Omron CX-Programmer project NewProject (CX-Programmer 9.73)

# PLC NewPLC1: CJ2M CPU12
I/O table (CPU CJ2M-CPU12): rack 0 slot 0 CJ1W-ID261; rack 0 slot 1 CJ1W-OD261; rack 0 slot 2 CJ1W-EIP21

## Global symbols (name address type ; comment)
AUTO 4030.00 BOOL  ; Auto
0.00 BOOL  ; (WP) SE Overload Product
0.01 BOOL  ; (HP) SE STOPPER SHIFTER
0.02 BOOL  ; (WP) SE STOPPER CHECKER 1
0.03 BOOL  ; (WP) SE STOPPER CHECKER 2
0.04 BOOL  ; (WP)SE NG PUSHER
0.05 BOOL  ; SE CHECKER 1
0.06 BOOL  ; SE CHECKER 2
0.07 BOOL  ; SE INPUT COUNT
0.08 BOOL  ; SE PRODUCT SHIFTER
0.09 BOOL  ; SE PRODUCT CHECKER 1
0.10 BOOL  ; SE PRODUCT CHECKER 2
0.11 BOOL  ; SE NG COUNT
0.12 BOOL  ; SE OUTPUT COUNT
0.13 BOOL  ; HP OVERLOAD PRODUCT
0.14 BOOL  ; WP OVERLOAD PRODUCT
0.15 BOOL  ; WP STOPPER SHIFTER
1.00 BOOL  ; WP STOPPER SHIFTER
1.01 BOOL  ; HP STOPPER CHECKER 1
1.02 BOOL  ; WP STOPPER CHECKER 1
1.03 BOOL  ; HP STOPPER CHECKER 2
1.04 BOOL  ; WP STOPPER CHECKER 2
1.05 BOOL  ; HP NG PUSHER
1.06 BOOL  ; WP NG PUSHER
1.07 BOOL  ; HP DOOR NG PRODUCT
1.08 BOOL  ; WP DOOR NG PRODUCT
1.09 BOOL  ; HP CHECKER 1
1.10 BOOL  ; WP CHECKER 1
1.11 BOOL  ; HP CHECKER 2
1.12 BOOL  ; WP CHECKER 2
1.13 BOOL  ; HP HORIZONTAL SHIFTER
1.14 BOOL  ; WP HORIZONTAL SHIFTER
1.15 BOOL  ; HP VERTICAL SHIFTER
2.00 BOOL  ; WP VERTICAL SHIFTER
2.01 BOOL  ; SE DOOR 1
2.02 BOOL  ; SE DOOR 2
2.03 BOOL  ; SE DOOR 3
2.04 BOOL  ; SE DOOR 4
2.05 BOOL  ; PB START 2
2.06 BOOL  ; PB START 1
2.07 BOOL  ; PB EXECUTE
2.08 BOOL  ; SE CHECKER 1 (2)
2.09 BOOL  ; SE CHECKER 1 (2)
2.15 BOOL  ; Pressure Sensor
300.00 BOOL  ; Hole Check Error
3070.00 BOOL  ; ALL HP TRANSFER
3070.01 BOOL  ; ALL HP CHECKER 1
3070.02 BOOL  ; ALL HP CHECKER 2
3070.03 BOOL  ; ALL HP NG EJECTOR
350.00 BOOL  ; U0_X_At_POS-0
350.01 BOOL  ; U0_X_At_POS-1
350.15 BOOL  ; U0_X_At_HOMEPOS
3.00 BOOL  ; AUTO BUTTON 1
3.01 BOOL  ; AUTO BUTTON 2
3.04 BOOL  ; DOOR SWITCH 1
3.05 BOOL  ; DOOR SWITCH 2
3.06 BOOL  ; DOOR SWITCH 3
3.07 BOOL  ; SE Minimum
3.08 BOOL  ; HP SEPARATOR 1
3.09 BOOL  ; HP SEPARATOR 2
3.10 BOOL  ; WP HOLDER
4000.00 BOOL  ; ON ON
4004.03 BOOL  ; FLG
4004.04 BOOL  ; BUSY
4004.05 BOOL  ; OR
4004.06 BOOL  ; RUN
4004.07 BOOL  ; ERROR
400.00 BOOL  ; TRANSFER_EMG_ALM
400.01 BOOL  ; CHECKER 1_EMG_ALM
400.02 BOOL  ; CHECKER 2 EMG_ALM
400.03 BOOL  ; NG EJECTOR_EMG_ALM
400.04 BOOL  ; 094 : Error Silinder NG Pusher
400.05 BOOL  ; 095 : Error Silinder Checker 1
400.06 BOOL  ; 096 : Error Silinder Checker 2
400.07 BOOL  ; 097 : Error Silinder Horizontral Shifter
400.08 BOOL  ; 098 : Error Silinder Vertical Shifter
400.09 BOOL  ; 099 : Error Silinder Door NG
400.15 BOOL  ; Transfer_EMG_Alarm
4010.00 BOOL  ; All Unit Ready
4010.01 BOOL  ; ALL CYL HP
4010.02 BOOL  ; NC Unit Error
4010.03 BOOL  ; ALL UNIT ORIGIN
4010.04 BOOL  ; ALL Manual OFF
4010.05 BOOL  ; ALL NO ALARM
4010.06 BOOL  ; Door Closed
4010.09 BOOL  ; Door Closed
4010.10 BOOL  ; READY Under RUN
4010.11 BOOL  ; READY AUTO START
4010.12 BOOL  ; ErrorReset Switch DU
401.00 BOOL  ; 090 : Error Silinder Holder Shifter (SE013/014) - Transfer
401.01 BOOL  ; 091 : Error Silinder Stopper Shifter (SE015/100) - Transfer
401.03 BOOL  ; 093 : Error Silinder Stopper Checker 2 (SE103/104) - Checking 2
401.04 BOOL  ; 094 : Error Silinder NG Pusher (SE105/106) - NG Ejector
401.05 BOOL  ; 095 : Error Silinder Checker 1 (SE109/110) - Checking 1
401.06 BOOL  ; 096 : Error Silinder Checker 2 (SE111/112) - Checking 2
401.07 BOOL  ; 097 : Error Silinder Horizontral Shifter (SE113/114) - Transfer
401.08 BOOL  ; 098 : Error Silinder Vertical Shifter (SE115/200) - Transfer
401.09 BOOL  ; 099 : Error Silinder Door NG (SE107/108) - NG Ejector
401.15 BOOL  ; Transfer ALM
4020.00 BOOL  ; Auto Index - Stop Lock
402.00 BOOL  ; 092 : Error Silinder Stopper Checker 1 (SE101/102) - Checking 1
402.00 BOOL  ; 092 : Error Silinder Stopper Checker 1
402.01 BOOL  ; 095 : Error Silinder Checker 1 (SE109/110) - Checking 1
402.15 BOOL  ; Checker 1 ALM
4030.00 BOOL  ; AUTO
4030.01 BOOL  ; STOP LOCK
4030.02 BOOL  ; STOP
4030.03 BOOL  ; Force STOP
4030.04 BOOL  ; Normal Run
4030.05 BOOL  ; Active Dry Run
4030.10 BOOL  ; Auto OFF
4031.00 BOOL  ; AUTO RUN PROCESS
4031.01 BOOL  ; SENSOR WORKING CHECK
4031.02 BOOL  ; SHIFT DATA UNIT WORK
4031.03 BOOL  ; START - AFTER CONFIRM
4031.04 BOOL  ; AUTO SAME START
4031.05 BOOL  ; AUTO DIFFERENT START
4031.06 BOOL  ; START Again
4031.07 BOOL  ; ReSTART Condition
4032.00 BOOL  ; AUTO - Transfer
4032.15 BOOL  ; FIN - Transfer
4033.00 BOOL  ; AUTO - Checker 1
4033.15 BOOL  ; FIN - Checker 1
4034.00 BOOL  ; AUTO - CHECKER 2
4034.15 BOOL  ; FIN - Checker 2
4035.00 BOOL  ; AUTO - NG EJECTOR
4035.04 BOOL  ; ACTIVE TYPE NON K
4035.05 BOOL  ; Active TYPE K
4035.15 BOOL  ; FIN - NG EJECTOR
4036.15 BOOL  ; FIN - Unloading
403.00 BOOL  ; 093 : Error Silinder Stopper Checker 2 (SE103/104) - Checking 2
403.01 BOOL  ; 096 : Error Silinder Checker 2 (SE111/112) - Checking 2
403.15 BOOL  ; Checker 2 ALM
4045.15 BOOL  ; ALL UNIT FINISH
4047.00 BOOL  ; Auto CL
4047.01 BOOL  ; Manu CL
4047.02 BOOL  ; RUN CLEAR LOAD
4047.03 BOOL  ; After Manual CL
404.00 BOOL  ; 094 : Error Silinder NG Pusher (SE105/106) - NG Ejector
404.01 BOOL  ; 099 : Error Silinder Door NG (SE107/108) - NG Ejector
404.09 BOOL  ; 099 : Error Silinder Door NG (SE107/108) - NG Ejector
404.15 BOOL  ; NG Ejector ALM
4050.00 BOOL  ; ALL EMPTY
4050.01 BOOL  ; ALL UNIT EMPTY
4050.02 BOOL  ; WORK - No Unit
4050.03 BOOL  ; WORK - Marking
4050.04 BOOL  ; WORK - No Unit
4050.05 BOOL  ; WORK - Unloading
4051.01 BOOL  ; All Unit Empty
4055.00 BOOL  ; Active Checker 1
4055.01 BOOL  ; Active No Unit
4055.02 BOOL  ; Active Checker 2
4055.03 BOOL  ; Active NG EJECTOR
4055.04 BOOL  ; Active NG STOPPER
4055.05 BOOL  ; Active Unloading
4056.00 BOOL  ; Active By Pass
405.00 BOOL  ; 095 : Error Silinder Checker 1
4060.10 BOOL  ; Fullwork
406.00 BOOL  ; 096 : Error Silinder Checker 2
4070.00 BOOL  ; EMG ALARM M/C
4070.01 BOOL  ; CYCLE ALARM M/C
4070.02 BOOL  ; NC UNIT ERROR
4076.03 BOOL  ; Active Marking No Part
407.00 BOOL  ; 097 : Error Silinder Horizontal Shifter
4080.00 BOOL  ; WAITING TIME
4081.00 BOOL  ; FULLWORK
4082.00 BOOL  ; BLOWING ON AFTER WAITING 2SEC
408.00 BOOL  ; 098 : Error Silinder Vertical Shifter
409.00 BOOL  ; 099 : Error Sillinder Door NG
4100.00 BOOL  ; Ready Transfer
4100.03 BOOL  ; Ready NG Stopper
4101.15 BOOL  ; DONE ORG Shifter Transfer
410.00 BOOL  ; Safety Door Alarm
4110.00 BOOL  ; POS 0 - Shifter Trasnfer
4110.01 BOOL  ; Pos 1 - Shifter Transfer
4110.15 BOOL  ; Home - Shifter Transfer
411.00 BOOL  ; 100 : Error Safety Door Front L (SE201) - Transfer
411.01 BOOL  ; 101 : Error Safety Door Front R (SE202) - Transfer
411.02 BOOL  ; 102 : Error Safety Door Back L (SE203) - Transfer
411.03 BOOL  ; 103 : Error Safety Door Back R (SE204) - Transfer
4120.00 BOOL  ; 1 Cycle Checking 1 (MANU)
4120.01 BOOL  ; Call Separator Seq
4120.05 BOOL  ; Ready Transfer
4121.00 BOOL  ; 1 Cycle Checking 2 (MANU)
4121.01 BOOL  ; Stopper On
4121.02 BOOL  ; Separator 1 On
4121.03 BOOL  ; Separator Off
4121.04 BOOL  ; Stopper Off
4121.11 BOOL  ; Stop Conv
4121.12 BOOL  ; On Conv
4121.15 BOOL  ; Finish Separator Seq
4122.00 BOOL  ; 1 Cycle Transfer (MANU)
4122.01 BOOL  ; Call Shifter
4123.00 BOOL  ; 1 Cycle NG Stopper (MANU)
4123.01 BOOL  ; Arm On
4123.02 BOOL  ; Separator 2 On
4123.03 BOOL  ; Shifter On
4123.04 BOOL  ; Arm Off
4123.05 BOOL  ; Separator 2 Off
4123.06 BOOL  ; Shifter Off
4123.10 BOOL  ; DONE - Transfer
4123.15 BOOL  ; Finish Shifter Seq
4124.00 BOOL  ; Status for Arm Down
4125.00 BOOL  ; 1 Cycle Checking NG
4126.00 BOOL  ; 1 Cycle NG Stopper (MANU)
4129.00 BOOL  ; 1 Cycle Process
412.00 BOOL  ; 104 : Error Low Air Pressure (SE215) - Transfer
4132.00 BOOL  ; MANUAL OFF
4140.00 BOOL  ; Anchor A_EMG_Error
4140.01 BOOL  ; Anchor A Error
4141.00 BOOL  ; 090 : Error Stopper (SE0100/0101) - Anchor A
4141.01 BOOL  ; 091 : Error Fwd/Bwd (SE0102/0103) - Anchor A
4141.02 BOOL  ; 092 : Error Rotary Esc (SE0104/0105) - Anchor A
4141.03 BOOL  ; 093 : Error Chuck PNP (SE0110) - Anchor A
4141.04 BOOL  ; 094 : Error Up/Dn Pusher (SE0111/0112) - Anchor A
4141.05 BOOL  ; 095 : Error Lift Case (SE0001/0002) - Anchor A
4141.06 BOOL  ; 096 : Error Holder Case (SE00114/00115) - Anchor A
4143.00 BOOL  ; 110 : Alarm Driver X Axis SMC - Anchor A
4143.01 BOOL  ; 111: Alarm Driver Y Axis SMC - Anchor A
4143.02 BOOL  ; 112 : Alarm Driver Rotary ARD K - Anchor A
4170.00 BOOL  ; Ready Transfer
4170.05 BOOL  ; Ready - Check HV
4172.10 BOOL  ; DONE - Check HV
4182.00 BOOL  ; Check HV Manu = OFF
4190.00 BOOL  ; Ready Transfer
4190.01 BOOL  ; Ready Checker 1
4190.02 BOOL  ; Ready Checker 2
4190.03 BOOL  ; Ready NG Stopper
4193.00 BOOL  ; Ready Transfer
4193.01 BOOL  ; Ready Checker 1
4193.02 BOOL  ; Ready Checker 2
4193.03 BOOL  ; Ready NG Stopper
4220.05 BOOL  ; Ready - Check CR
4221.15 BOOL  ; Finish Check CR
4222.10 BOOL  ; DONE - Check CR
4232.00 BOOL  ; Check CR Manu = OFF
4240.00 BOOL  ; Check CR_EMG_ALM
4240.01 BOOL  ; Check CR ALM
4270.05 BOOL  ; Ready - Marking
4282.00 BOOL  ; Marking Unit Manu = OFF
4290.00 BOOL  ; Marking Unit_EMG_ALM
4290.01 BOOL  ; Marking Unit ALM
4301.15 BOOL  ; DONE ORG Shifter Transfer
4320.05 BOOL  ; Ready - Unloading
4321.06 BOOL  ; Chuck Off
4324.00 BOOL  ; OK
4332.00 BOOL  ; Unloading Manu = OFF
4340.00 BOOL  ; Unloading_EMG_ALM
4340.01 BOOL  ; Unloading ALM
4390.00 BOOL  ; SafetyDoor_EMG_ALM
4390.01 BOOL  ; Safety Door ALM
4391.00 BOOL  ; Safety Door Front L
4391.01 BOOL  ; Safety Door Front C
4391.02 BOOL  ; Safety Door Front R
4391.03 BOOL  ; Safety Door Back L
4520.01 BOOL  ; Call START Check Hole 1
4520.02 BOOL  ; Call START Check Hole 2
4520.03 BOOL  ; Call NG
4520.15 BOOL  ; Finish Separator
4521.00 BOOL  ; START Check Hole 1
4521.01 BOOL  ; Holder 1 ON
4521.02 BOOL  ; Checker 1 DOWN
4521.03 BOOL  ; Checker 1 UP
4521.04 BOOL  ; Holder 1 OFF
4521.05 BOOL  ; CHECKER 2 ON
4521.06 BOOL  ; CHECKER 2 DOWN
4521.07 BOOL  ; CHECKER 2 UP
4521.08 BOOL  ; CHECKER 2 OFF
4521.10 BOOL  ; DONE - Checker 1
4521.15 BOOL  ; FINISH Check 1
4522.01 BOOL  ; Call Shifter
4523.00 BOOL  ; Start Shifter Seq
4523.01 BOOL  ; ARM VERTICAL ON
4523.02 BOOL  ; STOPPER ON
4523.03 BOOL  ; SHIFTER HORIZONTAL ON
4523.04 BOOL  ; ARM VERTICAL OFF
4523.05 BOOL  ; STOPPER OFF
4523.06 BOOL  ; SHIFTER HORIZONTAL OFF
4523.10 BOOL  ; DONE - Transfer
4523.15 BOOL  ; Finish Shifter Seq
4524.00 BOOL  ; START Check Hole 2
4524.01 BOOL  ; Holder 2 ON
4524.02 BOOL  ; Checker 2 DOWN
4524.03 BOOL  ; Checker 2 UP
4524.04 BOOL  ; Holder 2 OFF
4524.10 BOOL  ; DONE - Checker 2
4524.15 BOOL  ; FINISH Check 2
4525.00 BOOL  ; Start NG Seq
4525.01 BOOL  ; NG Door Down
4525.02 BOOL  ; NG Pusher ON
4525.03 BOOL  ; NG Pusher OFF
4525.04 BOOL  ; NG Door UP
4525.10 BOOL  ; DONE - NG EJECTOR
4525.15 BOOL  ; Finish NG Stopper Seq
4526.00 BOOL  ; Start NG Seq
4526.01 BOOL  ; NG Door DOWN
4526.02 BOOL  ; NG Pusher ON
4526.03 BOOL  ; NG Pusher OFF
4526.04 BOOL  ; NG Door UP
4526.15 BOOL  ; Finish NG Stopper Seq
4527.00 BOOL  ; Call Holder Seq
4527.01 BOOL  ; Holder On
4527.02 BOOL  ; Holder Off
4527.15 BOOL  ; Finish Seq Holder
4530.00 BOOL  ; START VISION 1 SEQ
4530.01 BOOL  ; MEASURE START VIS 1
4530.02 BOOL  ; MEASURE BUSY VIS 1
4530.03 BOOL  ; MEASURE FINISH VIS 1
4530.04 BOOL  ; JUDGE MEASURED
4530.15 BOOL  ; FINISH VISION 1
4531.00 BOOL  ; START VISION 2 SEQ
4531.01 BOOL  ; MEASURE START VIS 2
4531.02 BOOL  ; MEASURE BUSY VIS 2
4531.03 BOOL  ; MEASURE FINISH VIS 2
4531.04 BOOL  ; JUDGE MEASURED VIS 2
4531.05 BOOL  ; HOLDER OPEN VIS 2
4531.15 BOOL  ; FINISH VISION 2
4560.00 BOOL  ; Manual Transfer Active
4560.01 BOOL  ; Manual Checking 1 Active
4560.02 BOOL  ; Manual Checking 2 Active
4560.03 BOOL  ; Manual NG Ejector ACTIVE
4626.00 BOOL  ; Display OK/NG
4670.00 BOOL  ; PASSWORD CORRECT
4671.00 BOOL  ; Password SHOWUP
468.00 BOOL  ; TES
4725.00 BOOL  ; BLOWING ON
4725.01 BOOL  ; RUN 1x
4800.00 BOOL  ; Ready Transfer
4.00 BOOL  ; Silinder Overload Product
4.01 BOOL  ; Silinder Stopper Shifter
4.02 BOOL  ; Silinder Stopper Checker 1
4.03 BOOL  ; Silinder Stopper Checker 2
4.04 BOOL  ; Silinder NG Pusher
4.05 BOOL  ; Silinder Checker 1 DOWN
4.06 BOOL  ; Silinder Checker 1 UP
4.07 BOOL  ; Silinder Horizontal Shifter
4.08 BOOL  ; Silinder Vertical Shifter
4.09 BOOL  ; Silinder Door NG Product
4.10 BOOL  ; Buzzer
4.11 BOOL  ; Lamp PB Execute
4.12 BOOL  ; Lamp PB Start 1
4.13 BOOL  ; Air Pressure
4.14 BOOL  ; Lamp Red
4.15 BOOL  ; Lamp Green
5001.00 BOOL  ; Home Marking
500.00 BOOL  ; SILINDER OVERLOAD PRODUCT
500.01 BOOL  ; SILINDER STOPPER SHIFTER
500.02 BOOL  ; SILINDER STOPPER CHECKER 1
500.03 BOOL  ; SILINDER STOPPER CHECKER 2
500.04 BOOL  ; SILINDER NG PUSHER
500.05 BOOL  ; CHECKER 1 U/D
500.06 BOOL  ; CHECKER 2 U/D
500.07 BOOL  ; SILINDER HORIZONTAL SHIFTER
500.08 BOOL  ; SILINDER VERTICAL SHIFTER
500.09 BOOL  ; SILINDER DOOR NG PRODUCT
500.10 BOOL  ; BUZZER
500.11 BOOL  ; LAMP PB EXECUTE
500.12 BOOL  ; LAMP PB START 1
500.13 BOOL  ; AIR PRESSURE START
500.14 BOOL  ; LAMP RED
500.15 BOOL  ; LAMP GREEN
5010.00 BOOL  ; Reset
501.00 BOOL  ; MOTOR 1
501.01 BOOL  ; MOTOR 2
501.02 BOOL  ; Checker 2 DOWN
501.03 BOOL  ; Checker 2 UP
501.04 BOOL  ; Overload
501.05 BOOL  ; STOP
501.07 BOOL  ; Pressure 1
501.10 BOOL  ; MOTOR 2
501.15 BOOL  ; BLOWING
505.00 BOOL  ; Disable Marking
5.00 BOOL  ; Motor 1
5.01 BOOL  ; Motor 2
5.02 BOOL  ; Silinder Checker 2 DOWN
5.03 BOOL  ; Silinder Checker 2 UP
5.14 BOOL  ; NG DOOR LOCK
5.15 BOOL  ; BLOWING
645.00 BOOL  ; Reset Man CL
6.00 BOOL  ; WAITING TIME
700.00 BOOL  ; NG Check 1
70.00 BOOL  ; NG CHECK 1
760.00 BOOL  ; U/D  Checker 1
761.00 BOOL  ; U/D Checker 2
765.00 BOOL  ; Target Achieve
766.00 BOOL  ; NO TARGET
87.00 BOOL  ; Latch Main
D110 CHANNEL  ; Hasil Perhitungan EFF M/C
D11000 CHANNEL  ; Total Alarm Time
D120 CHANNEL  ; TOTAL OUTPUT OK+NG
D123 CHANNEL  ; CT M/C on Process
D124 CHANNEL  ; Output Target CT 1.5
D131 CHANNEL  ; Theoretical CT
D160 CHANNEL  ; YIELD RATIO
D18251 CHANNEL  ; M/C Cycle Time
D18270 CHANNEL  ; Output
D18271 CHANNEL  ; Input
D18284 CHANNEL  ; M/C Efficiency
D19299 CHANNEL  ; $?St$Bk?_#[6] / $?St$Bk?_#[6]
D19900 CHANNEL  ; Auto Run (second)
D19999 CHANNEL  ; $?St$Bk?_#[7] / $?St$Bk?_#[7]
D20000 CHANNEL  ; Total Alarm
D21100 CHANNEL  ; STOP TIME (second)
D21200 CHANNEL  ; ALARM TIME (second)
D21300 CHANNEL  ; OUTPUT OK
D21400 CHANNEL  ; WAITING TIME ( SEC )
D21500 CHANNEL  ; OUTPUT NG
D21600 CHANNEL  ; FULLWORK TIME (SEC)
D250 CHANNEL  ; TYPE
D4000 CHANNEL  ; OVERLOAD
D4002 CHANNEL  ; STOPPER
D4004 CHANNEL  ; STOPPER CHECKER 1
D4006 CHANNEL  ; STOPPER CHECKER 2
D4008 CHANNEL  ; NG PUSHER
D4010 CHANNEL  ; CHECKER 1 U/D
D4012 CHANNEL  ; Horizontal Shifter
D4014 CHANNEL  ; Vertical Shifter
D4016 CHANNEL  ; DOOR NG
D4018 CHANNEL  ; CHECKER 2 U/D
D4020 CHANNEL  ; Overload
E0.07 BOOL  ; SE Part 2
H10.00 BOOL  ; WORK - Checking 1
H10.01 BOOL  ; WORK - No Unit
H10.02 BOOL  ; WORK - Checker 2
H10.03 BOOL  ; WORK - NG Stopper
H10.04 BOOL  ; WORK - NG STOPPER
H14.00 BOOL  ; Enable Unit Checker 1
H14.01 BOOL  ; Enable Unit Checker 2
H14.02 BOOL  ; Enable Unit NG Stopper
H14.04 BOOL  ; Enable Unit Unloading
H18.00 BOOL  ; TYPE K
H18.01 BOOL  ; TYPE NON-K
H20.00 BOOL  ; Data Part In
H21.00 BOOL  ; OUTPUT NG
H25.00 BOOL  ; Active By Pass
H25.01 BOOL  ; NORMAL MODE
H25.02 BOOL  ; DRY RUN MODE
H70.00 BOOL  ; NG CHECK 1
H70.01 BOOL  ; NG CHECK 2
H72.00 BOOL  ; NG CHECK 1 (2)
T0060 BOOL  ; TIM ERROR
T0125 BOOL  ; RESET 1 SEC
T0200 BOOL  ; WAITING TIME
T0520 BOOL  ; Auto Button
T0521 BOOL  ; Auto Index Delay Finish
T0530 BOOL  ; UNIT WORKING AFTER CONFIRM (Dont ZERO)
T0531 BOOL  ; Delay for Start Again
T0533 BOOL  ; Time START CL
T0534 BOOL  ; DIFFERENT START
T0750 BOOL  ; Delay Checker 1
T0751 BOOL  ; Delay Checker 2
W0.00 BOOL  ; (WP)SE Overload Product
W0.01 BOOL  ; (HP)SE STOPPER SHIFTER
W0.02 BOOL  ; (WP)SE STOPPER CHECKER 1
W0.03 BOOL  ; (WP)SE STOPPER CHECKER 2
W0.04 BOOL  ; (WP)SE NG PUSHER
W0.05 BOOL  ; SE CHECKER 1
W0.06 BOOL  ; SE CHECKER 2
W0.07 BOOL  ; SE INPUT COUNT
W0.08 BOOL  ; SE PRODUCT SHIFTER
W0.09 BOOL  ; SE PRODUCT CHECKER 1
W0.10 BOOL  ; SE PRODUCT  CHECKER 2
W0.11 BOOL  ; SE NG COUNT
W0.12 BOOL  ; SE OUTPUT COUNT
W0.13 BOOL  ; HP SILINDER OVERLOAD PRODUCT
W0.14 BOOL  ; WP SILINDER OVERLOAD PRODUCT
W0.15 BOOL  ; WP SILINDER STOPPER SHIFTER
W110.00 BOOL  ; PB SILINDER OVERLOAD PRODUCT
W110.01 BOOL  ; PB SILINDER STOPPER SHIFTER
W110.02 BOOL  ; PB SILINDER STOPPER CHECKER 1
W110.03 BOOL  ; PB SILINDER STOPPER CHECKER 2
W110.04 BOOL  ; PB SILINDER NG PUSHER
W110.05 BOOL  ; PB SILINDER CHECKER 1
W110.06 BOOL  ; PB SILINDER CHECKER 2
W110.07 BOOL  ; PB SILINDER HORIZONTAL SHIFTER
W110.08 BOOL  ; PB SILINDER VERTICAL SHIFTER
W110.09 BOOL  ; PB SILINDER DOOR NG PRODUCT
W110.10 BOOL  ; PB BUZZER
W110.11 BOOL  ; PB LAMP PB EXECUTE
W110.12 BOOL  ; PB LAMP PB START 1
W110.13 BOOL  ; PB AIR PRESSURE
W110.14 BOOL  ; PB LAMP RED
W110.15 BOOL  ; PB LAMP GREEN
W111.00 BOOL  ; PB MOTOR 1
W111.01 BOOL  ; PB MOTOR 2
W111.02 BOOL  ; PB BLOWING
W111.10 BOOL  ; PB MOTOR 2
W120.00 BOOL  ; NS 1 Cycle Checking 1 (MANU)
W121.00 BOOL  ; NS 1 Cycle Checking 2 (MANU)
W122.00 BOOL  ; NS 1 Cycle Transfer  (MANU)
W123.00 BOOL  ; NS 1 Cycle NG Stopper (MANU)
W15.00 BOOL  ; NB By Pass M/C
W1.00 BOOL  ; WP SILINDER STOPPER SHIFTER
W1.01 BOOL  ; HP SILINDER STOPPER CHECKER 1
W1.02 BOOL  ; WP SILINDER STOPPER CHECKER 1
W1.03 BOOL  ; HP SILINDER STOPPER CHECKER 2
W1.04 BOOL  ; WP SILINDER STOPPER CHECKER 2
W1.05 BOOL  ; HP SILINDER NG PUSHER
W1.06 BOOL  ; WP SILINDER NG PUSHER
W1.07 BOOL  ; HP SILINDER DOOR NG PRODUCT
W1.08 BOOL  ; WP SILINDER DOOR NG PRODUCT
W1.09 BOOL  ; HP SILINDER CHECKER 1
W1.10 BOOL  ; WP SILINDER CHECKER 1
W1.11 BOOL  ; HP SILINDER CHECKER 2
W1.12 BOOL  ; WP SILINDER CHECKER 2
W1.13 BOOL  ; HP SILINDER HORIZONTAL SHIFTER
W1.14 BOOL  ; WP SILINDER HORIZONTAL SHIFTER
W1.15 BOOL  ; HP SILINDER VERTICAL SHIFTER
W20.00 BOOL  ; MAIN SW
W2.00 BOOL  ; WP SILINDER VERTICAL SHIFTER
W2.01 BOOL  ; SE SAFETY DOOR 1 (Front L)
W2.02 BOOL  ; SE SAFETY DOOR 2 (Front R)
W2.03 BOOL  ; SE SAFETYDOOR 3 (Back L)
W2.04 BOOL  ; SE SAFETYDOOR 4 (Back R)
W2.05 BOOL  ; PB START 2
W2.06 BOOL  ; PB START 1
W2.07 BOOL  ; PB EXECUTE
W2.08 BOOL  ; SE CHECKER 1 (2)
W2.09 BOOL  ; SE CHECKER 1 (2)
W2.15 BOOL  ; PRESSURE SENSOR
W30.00 BOOL  ; NS AUTO RUN
W30.03 BOOL  ; NS Normal Run
W30.04 BOOL  ; NS Dry Run
W30.05 BOOL  ; Manu Clear Load
W35.03 BOOL  ; NS TYPE NON K
W35.04 BOOL  ; NS TYPE K
W3.00 BOOL  ; VIS 1 FLG
W3.01 BOOL  ; VIS1 BUSY
W3.02 BOOL  ; VIS1 OR
W3.03 BOOL  ; VIS 1 RUN
W3.04 BOOL  ; VIS 1 ERROR
W3.05 BOOL  ; VIS2 FLG
W3.06 BOOL  ; VIS2 BUSY
W3.07 BOOL  ; VIS2 OR
W3.08 BOOL  ; VIS2 RUN
W3.09 BOOL  ; VIS2 ERROR
W50.00 BOOL  ; NS Checking 1 Active
W50.01 BOOL  ; NS Checking 2 Active
W50.02 BOOL  ; NS NG Active
W50.03 BOOL  ; NS Checking Active
W50.04 BOOL  ; NS Take Out Active
W52.01 BOOL  ; Reset Start Interlock
W60.00 BOOL  ; STOP
W6.00 BOOL  ; WAITING TIME
W70.00 BOOL  ; NS Reset ALM
W70.01 BOOL  ; Reset Record
W70.02 BOOL  ; Reset Time Record
W71.00 BOOL  ; DISPLAY OK/NG
ERROR_RST 4010.12 BOOL  ; ErrorReset Switch DU
EXECUTE W10.00 BOOL
OFF CF114 BOOL  ; ALWAYS OFF
ON CF113 BOOL  ; ALWAYS ON
ON_ON 4000.00 BOOL
RESET W70.00 BOOL  ; NS Reset ALM
RST_RECORD W70.01 BOOL  ; Reset Record

## Program Main_Control (cyclic task 0)
Local symbols
First_On BOOL
ON CF113 BOOL
P_OFF BOOL
on BOOL

### Section Input

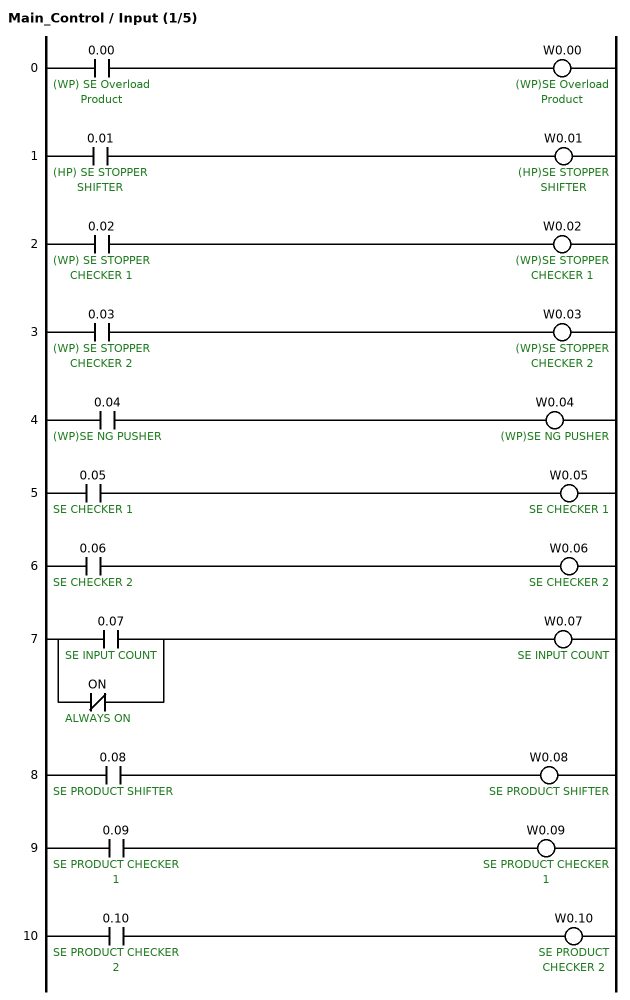
; rung 0
LD 0.00  ; (WP) SE Overload Product
OUT W0.00  ; (WP)SE Overload Product
; rung 1
LD 0.01  ; (HP) SE STOPPER SHIFTER
OUT W0.01  ; (HP)SE STOPPER SHIFTER
; rung 2
LD 0.02  ; (WP) SE STOPPER CHECKER 1
OUT W0.02  ; (WP)SE STOPPER CHECKER 1
; rung 3
LD 0.03  ; (WP) SE STOPPER CHECKER 2
OUT W0.03  ; (WP)SE STOPPER CHECKER 2
; rung 4
LD 0.04  ; (WP)SE NG PUSHER
OUT W0.04  ; (WP)SE NG PUSHER
; rung 5
LD 0.05  ; SE CHECKER 1
OUT W0.05  ; SE CHECKER 1
; rung 6
LD 0.06  ; SE CHECKER 2
OUT W0.06  ; SE CHECKER 2
; rung 7
LD 0.07  ; SE INPUT COUNT
ORNOT ON  ; ALWAYS ON
OUT W0.07  ; SE INPUT COUNT
; rung 8
LD 0.08  ; SE PRODUCT SHIFTER
OUT W0.08  ; SE PRODUCT SHIFTER
; rung 9
LD 0.09  ; SE PRODUCT CHECKER 1
OUT W0.09  ; SE PRODUCT CHECKER 1
; rung 10
LD 0.10  ; SE PRODUCT CHECKER 2
OUT W0.10  ; SE PRODUCT  CHECKER 2

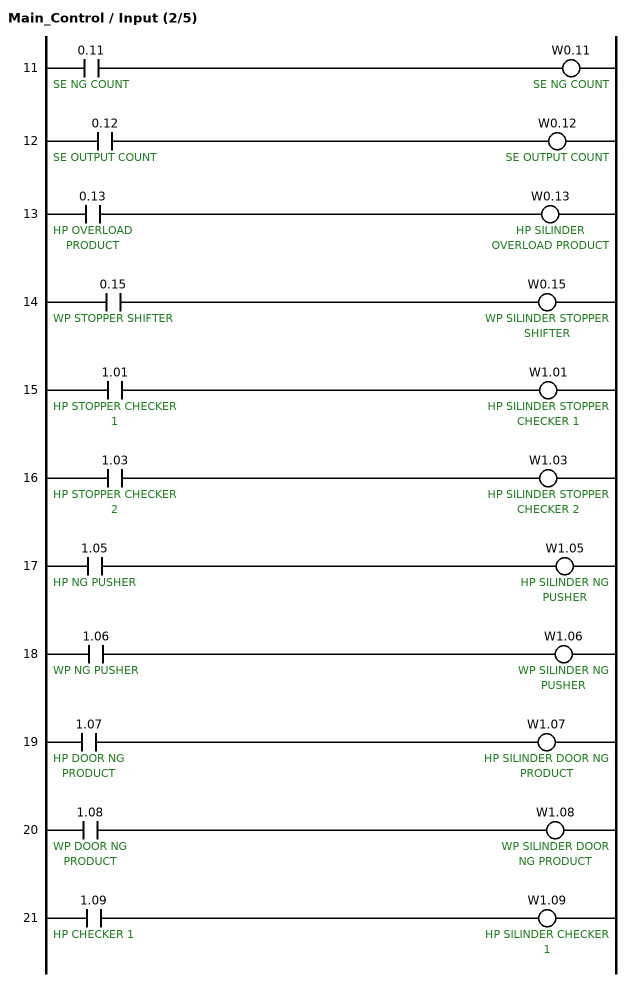
; rung 11
LD 0.11  ; SE NG COUNT
OUT W0.11  ; SE NG COUNT
; rung 12
LD 0.12  ; SE OUTPUT COUNT
OUT W0.12  ; SE OUTPUT COUNT
; rung 13
LD 0.13  ; HP OVERLOAD PRODUCT
OUT W0.13  ; HP SILINDER OVERLOAD PRODUCT
; rung 14
LD 0.15  ; WP STOPPER SHIFTER
OUT W0.15  ; WP SILINDER STOPPER SHIFTER
; rung 15
LD 1.01  ; HP STOPPER CHECKER 1
OUT W1.01  ; HP SILINDER STOPPER CHECKER 1
; rung 16
LD 1.03  ; HP STOPPER CHECKER 2
OUT W1.03  ; HP SILINDER STOPPER CHECKER 2
; rung 17
LD 1.05  ; HP NG PUSHER
OUT W1.05  ; HP SILINDER NG PUSHER
; rung 18
LD 1.06  ; WP NG PUSHER
OUT W1.06  ; WP SILINDER NG PUSHER
; rung 19
LD 1.07  ; HP DOOR NG PRODUCT
OUT W1.07  ; HP SILINDER DOOR NG PRODUCT
; rung 20
LD 1.08  ; WP DOOR NG PRODUCT
OUT W1.08  ; WP SILINDER DOOR NG PRODUCT
; rung 21
LD 1.09  ; HP CHECKER 1
OUT W1.09  ; HP SILINDER CHECKER 1

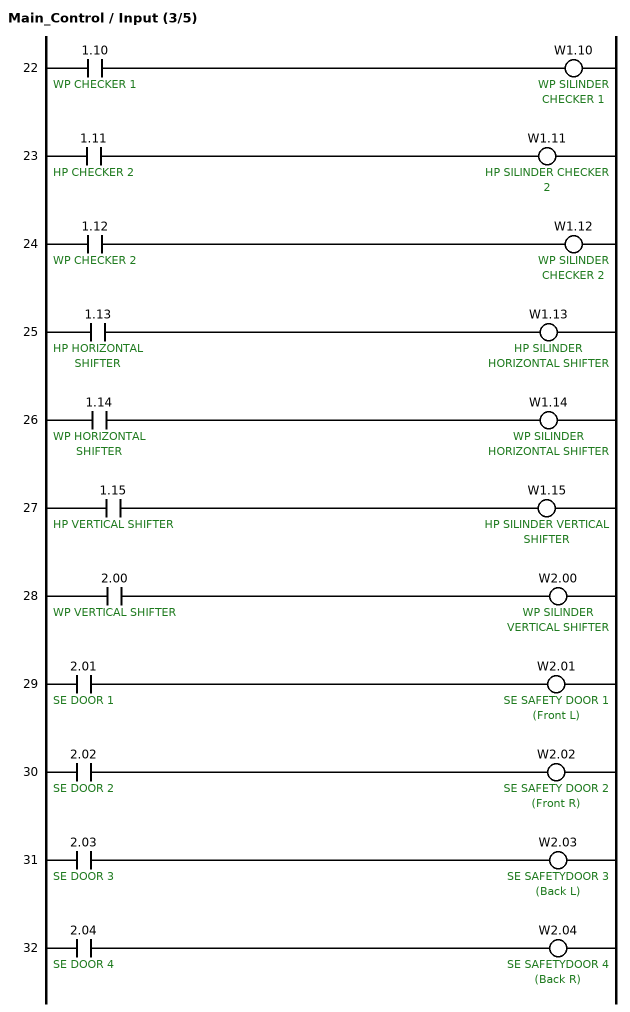
; rung 22
LD 1.10  ; WP CHECKER 1
OUT W1.10  ; WP SILINDER CHECKER 1
; rung 23
LD 1.11  ; HP CHECKER 2
OUT W1.11  ; HP SILINDER CHECKER 2
; rung 24
LD 1.12  ; WP CHECKER 2
OUT W1.12  ; WP SILINDER CHECKER 2
; rung 25
LD 1.13  ; HP HORIZONTAL SHIFTER
OUT W1.13  ; HP SILINDER HORIZONTAL SHIFTER
; rung 26
LD 1.14  ; WP HORIZONTAL SHIFTER
OUT W1.14  ; WP SILINDER HORIZONTAL SHIFTER
; rung 27
LD 1.15  ; HP VERTICAL SHIFTER
OUT W1.15  ; HP SILINDER VERTICAL SHIFTER
; rung 28
LD 2.00  ; WP VERTICAL SHIFTER
OUT W2.00  ; WP SILINDER VERTICAL SHIFTER
; rung 29
LD 2.01  ; SE DOOR 1
OUT W2.01  ; SE SAFETY DOOR 1 (Front L)
; rung 30
LD 2.02  ; SE DOOR 2
OUT W2.02  ; SE SAFETY DOOR 2 (Front R)
; rung 31
LD 2.03  ; SE DOOR 3
OUT W2.03  ; SE SAFETYDOOR 3 (Back L)
; rung 32
LD 2.04  ; SE DOOR 4
OUT W2.04  ; SE SAFETYDOOR 4 (Back R)

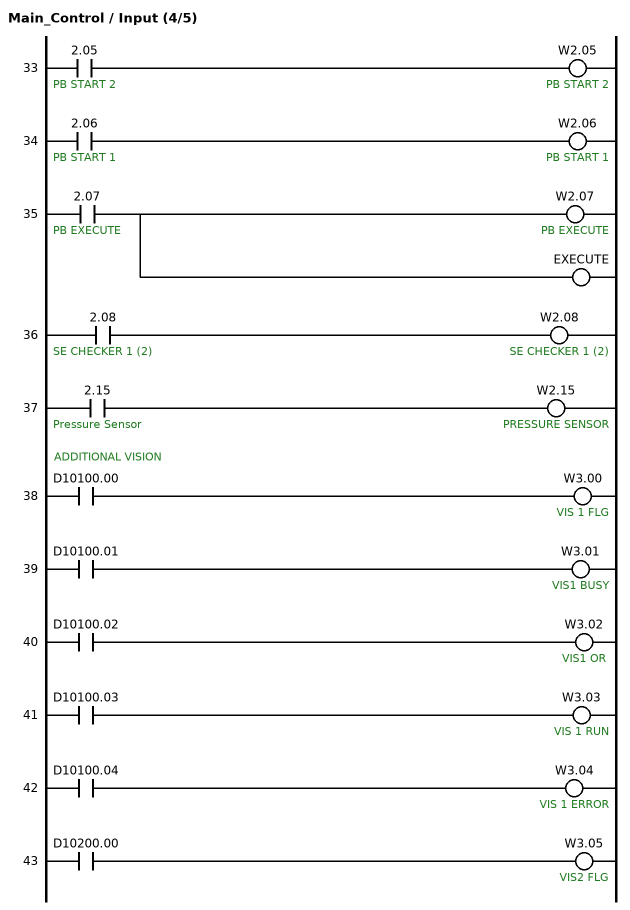
; rung 33
LD 2.05  ; PB START 2
OUT W2.05  ; PB START 2
; rung 34
LD 2.06  ; PB START 1
OUT W2.06  ; PB START 1
; rung 35
LD 2.07  ; PB EXECUTE
OUT W2.07  ; PB EXECUTE
OUT EXECUTE
; rung 36
LD 2.08  ; SE CHECKER 1 (2)
OUT W2.08  ; SE CHECKER 1 (2)
; rung 37
LD 2.15  ; Pressure Sensor
OUT W2.15  ; PRESSURE SENSOR
; rung 38: ADDITIONAL VISION
LD D10100.00
OUT W3.00  ; VIS 1 FLG
; rung 39
LD D10100.01
OUT W3.01  ; VIS1 BUSY
; rung 40
LD D10100.02
OUT W3.02  ; VIS1 OR
; rung 41
LD D10100.03
OUT W3.03  ; VIS 1 RUN
; rung 42
LD D10100.04
OUT W3.04  ; VIS 1 ERROR
; rung 43
LD D10200.00
OUT W3.05  ; VIS2 FLG

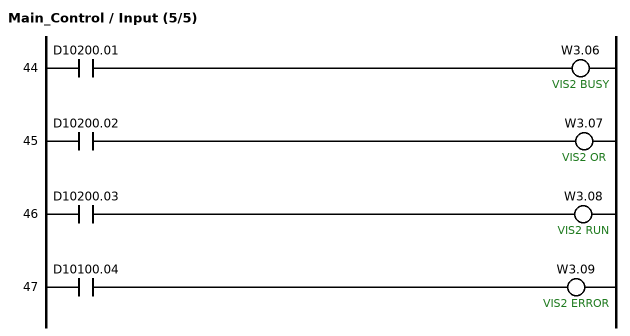
; rung 44
LD D10200.01
OUT W3.06  ; VIS2 BUSY
; rung 45
LD D10200.02
OUT W3.07  ; VIS2 OR
; rung 46
LD D10200.03
OUT W3.08  ; VIS2 RUN
; rung 47
LD D10100.04
OUT W3.09  ; VIS2 ERROR

### Section Output

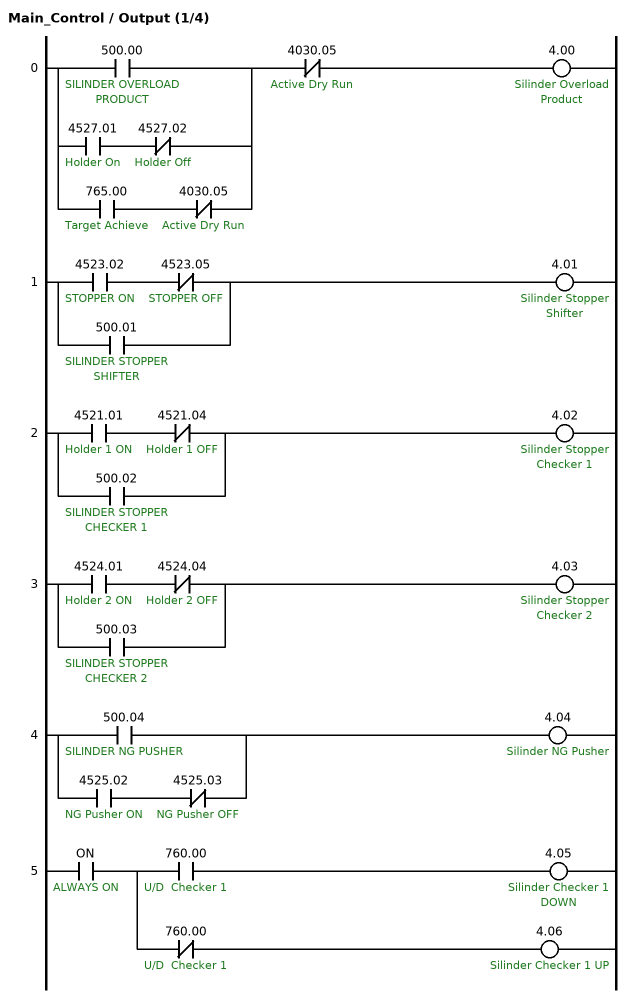
; rung 0
LD 500.00  ; SILINDER OVERLOAD PRODUCT
LD 4527.01  ; Holder On
ANDNOT 4527.02  ; Holder Off
ORLD
LD 765.00  ; Target Achieve
ANDNOT 4030.05  ; Active Dry Run
ORLD
ANDNOT 4030.05  ; Active Dry Run
OUT 4.00  ; Silinder Overload Product
; rung 1
LD 4523.02  ; STOPPER ON
ANDNOT 4523.05  ; STOPPER OFF
OR 500.01  ; SILINDER STOPPER SHIFTER
OUT 4.01  ; Silinder Stopper Shifter
; rung 2
LD 4521.01  ; Holder 1 ON
ANDNOT 4521.04  ; Holder 1 OFF
OR 500.02  ; SILINDER STOPPER CHECKER 1
OUT 4.02  ; Silinder Stopper Checker 1
; rung 3
LD 4524.01  ; Holder 2 ON
ANDNOT 4524.04  ; Holder 2 OFF
OR 500.03  ; SILINDER STOPPER CHECKER 2
OUT 4.03  ; Silinder Stopper Checker 2
; rung 4
LD 500.04  ; SILINDER NG PUSHER
LD 4525.02  ; NG Pusher ON
ANDNOT 4525.03  ; NG Pusher OFF
ORLD
OUT 4.04  ; Silinder NG Pusher
; rung 5
LD ON  ; ALWAYS ON
OUT TR0
AND 760.00  ; U/D  Checker 1
OUT 4.05  ; Silinder Checker 1 DOWN
LD TR0
ANDNOT 760.00  ; U/D  Checker 1
OUT 4.06  ; Silinder Checker 1 UP

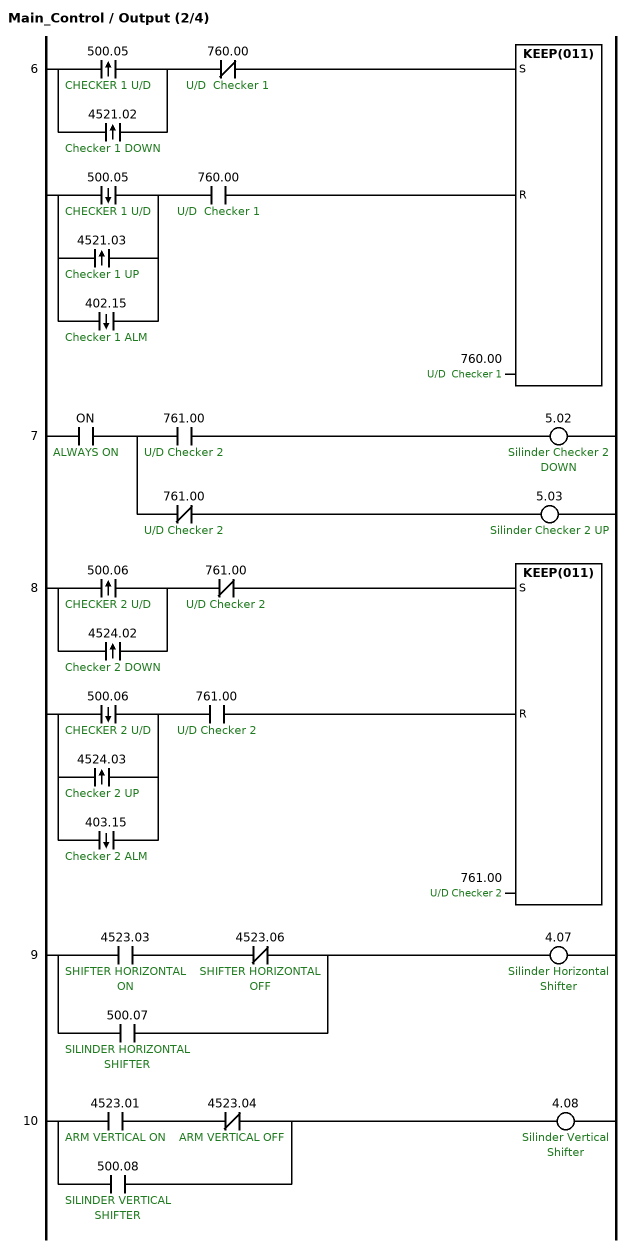
; rung 6
@LD 500.05  ; CHECKER 1 U/D
@OR 4521.02  ; Checker 1 DOWN
ANDNOT 760.00  ; U/D  Checker 1
%LD 500.05  ; CHECKER 1 U/D
@OR 4521.03  ; Checker 1 UP
%OR 402.15  ; Checker 1 ALM
AND 760.00  ; U/D  Checker 1
KEEP(011) 760.00  ; U/D  Checker 1
; rung 7
LD ON  ; ALWAYS ON
OUT TR0
AND 761.00  ; U/D Checker 2
OUT 5.02  ; Silinder Checker 2 DOWN
LD TR0
ANDNOT 761.00  ; U/D Checker 2
OUT 5.03  ; Silinder Checker 2 UP
; rung 8
@LD 500.06  ; CHECKER 2 U/D
@OR 4524.02  ; Checker 2 DOWN
ANDNOT 761.00  ; U/D Checker 2
%LD 500.06  ; CHECKER 2 U/D
@OR 4524.03  ; Checker 2 UP
%OR 403.15  ; Checker 2 ALM
AND 761.00  ; U/D Checker 2
KEEP(011) 761.00  ; U/D Checker 2
; rung 9
LD 4523.03  ; SHIFTER HORIZONTAL ON
ANDNOT 4523.06  ; SHIFTER HORIZONTAL OFF
OR 500.07  ; SILINDER HORIZONTAL SHIFTER
OUT 4.07  ; Silinder Horizontal Shifter
; rung 10
LD 4523.01  ; ARM VERTICAL ON
ANDNOT 4523.04  ; ARM VERTICAL OFF
OR 500.08  ; SILINDER VERTICAL SHIFTER
OUT 4.08  ; Silinder Vertical Shifter

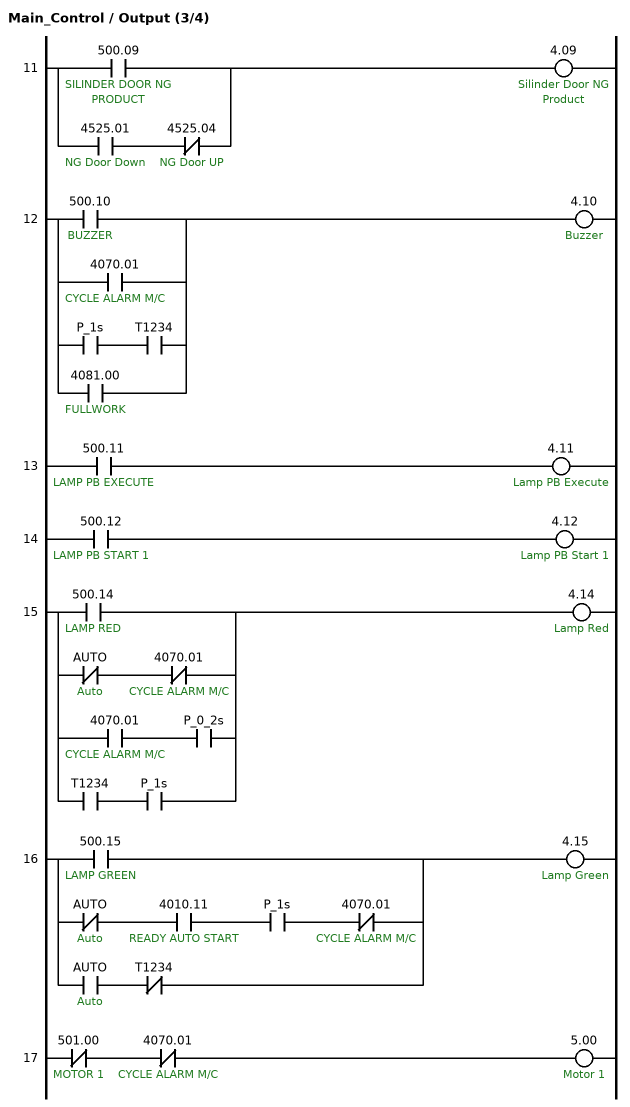
; rung 11
LD 500.09  ; SILINDER DOOR NG PRODUCT
LD 4525.01  ; NG Door Down
ANDNOT 4525.04  ; NG Door UP
ORLD
OUT 4.09  ; Silinder Door NG Product
; rung 12
LD 500.10  ; BUZZER
OR 4070.01  ; CYCLE ALARM M/C
LD P_1s
AND T1234
ORLD
OR 4081.00  ; FULLWORK
OUT 4.10  ; Buzzer
; rung 13
LD 500.11  ; LAMP PB EXECUTE
OUT 4.11  ; Lamp PB Execute
; rung 14
LD 500.12  ; LAMP PB START 1
OUT 4.12  ; Lamp PB Start 1
; rung 15
LD 500.14  ; LAMP RED
LDNOT AUTO  ; Auto
ANDNOT 4070.01  ; CYCLE ALARM M/C
ORLD
LD 4070.01  ; CYCLE ALARM M/C
AND P_0_2s
ORLD
LD T1234
AND P_1s
ORLD
OUT 4.14  ; Lamp Red
; rung 16
LD 500.15  ; LAMP GREEN
LDNOT AUTO  ; Auto
AND 4010.11  ; READY AUTO START
AND P_1s
ANDNOT 4070.01  ; CYCLE ALARM M/C
ORLD
LD AUTO  ; Auto
ANDNOT T1234
ORLD
OUT 4.15  ; Lamp Green
; rung 17
LDNOT 501.00  ; MOTOR 1
ANDNOT 4070.01  ; CYCLE ALARM M/C
OUT 5.00  ; Motor 1

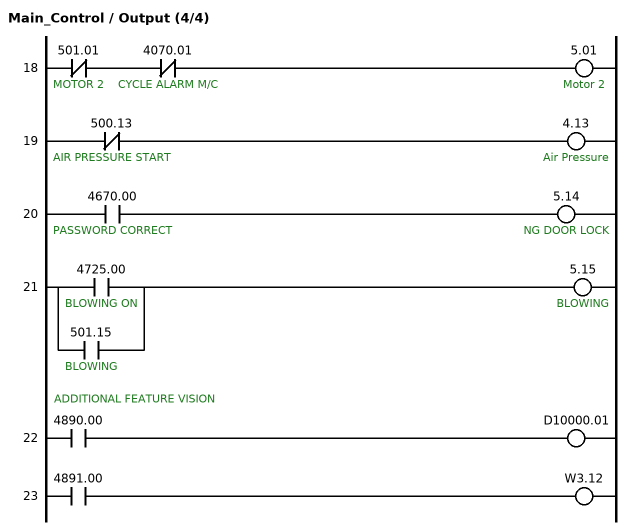
; rung 18
LDNOT 501.01  ; MOTOR 2
ANDNOT 4070.01  ; CYCLE ALARM M/C
OUT 5.01  ; Motor 2
; rung 19
LDNOT 500.13  ; AIR PRESSURE START
OUT 4.13  ; Air Pressure
; rung 20
LD 4670.00  ; PASSWORD CORRECT
OUT 5.14  ; NG DOOR LOCK
; rung 21
LD 4725.00  ; BLOWING ON
OR 501.15  ; BLOWING
OUT 5.15  ; BLOWING
; rung 22: ADDITIONAL FEATURE VISION
LD 4890.00
OUT D10000.01
; rung 23
LD 4891.00
OUT W3.12

### Section Manual

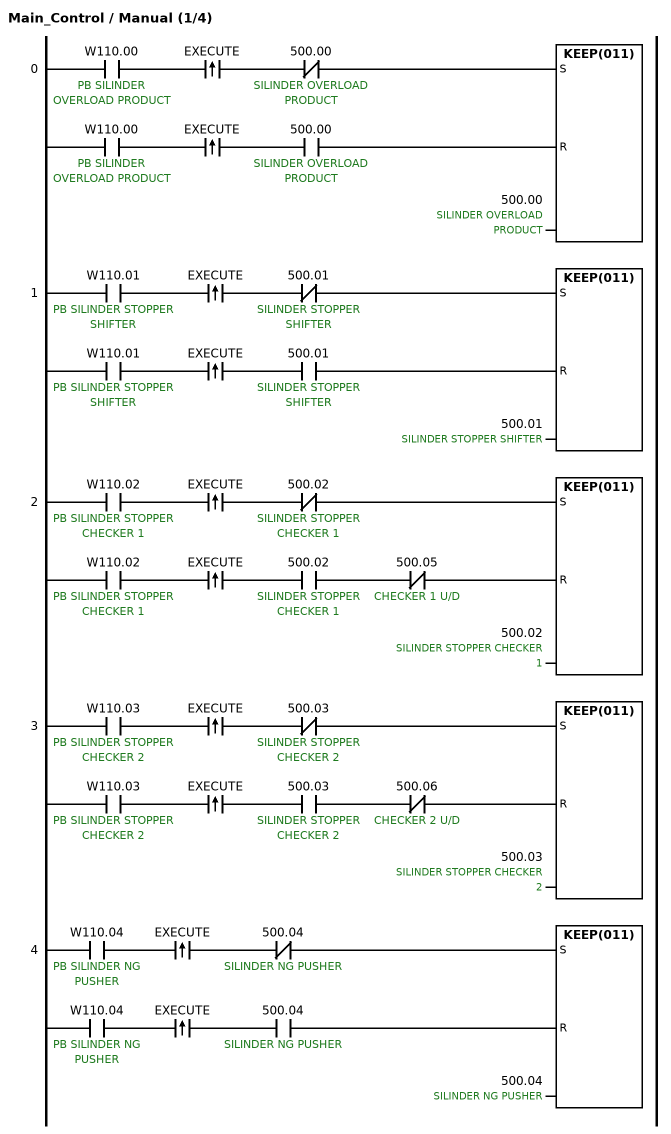
; rung 0
LD W110.00  ; PB SILINDER OVERLOAD PRODUCT
@AND EXECUTE
ANDNOT 500.00  ; SILINDER OVERLOAD PRODUCT
LD W110.00  ; PB SILINDER OVERLOAD PRODUCT
@AND EXECUTE
AND 500.00  ; SILINDER OVERLOAD PRODUCT
KEEP(011) 500.00  ; SILINDER OVERLOAD PRODUCT
; rung 1
LD W110.01  ; PB SILINDER STOPPER SHIFTER
@AND EXECUTE
ANDNOT 500.01  ; SILINDER STOPPER SHIFTER
LD W110.01  ; PB SILINDER STOPPER SHIFTER
@AND EXECUTE
AND 500.01  ; SILINDER STOPPER SHIFTER
KEEP(011) 500.01  ; SILINDER STOPPER SHIFTER
; rung 2
LD W110.02  ; PB SILINDER STOPPER CHECKER 1
@AND EXECUTE
ANDNOT 500.02  ; SILINDER STOPPER CHECKER 1
LD W110.02  ; PB SILINDER STOPPER CHECKER 1
@AND EXECUTE
AND 500.02  ; SILINDER STOPPER CHECKER 1
ANDNOT 500.05  ; CHECKER 1 U/D
KEEP(011) 500.02  ; SILINDER STOPPER CHECKER 1
; rung 3
LD W110.03  ; PB SILINDER STOPPER CHECKER 2
@AND EXECUTE
ANDNOT 500.03  ; SILINDER STOPPER CHECKER 2
LD W110.03  ; PB SILINDER STOPPER CHECKER 2
@AND EXECUTE
AND 500.03  ; SILINDER STOPPER CHECKER 2
ANDNOT 500.06  ; CHECKER 2 U/D
KEEP(011) 500.03  ; SILINDER STOPPER CHECKER 2
; rung 4
LD W110.04  ; PB SILINDER NG PUSHER
@AND EXECUTE
ANDNOT 500.04  ; SILINDER NG PUSHER
LD W110.04  ; PB SILINDER NG PUSHER
@AND EXECUTE
AND 500.04  ; SILINDER NG PUSHER
KEEP(011) 500.04  ; SILINDER NG PUSHER

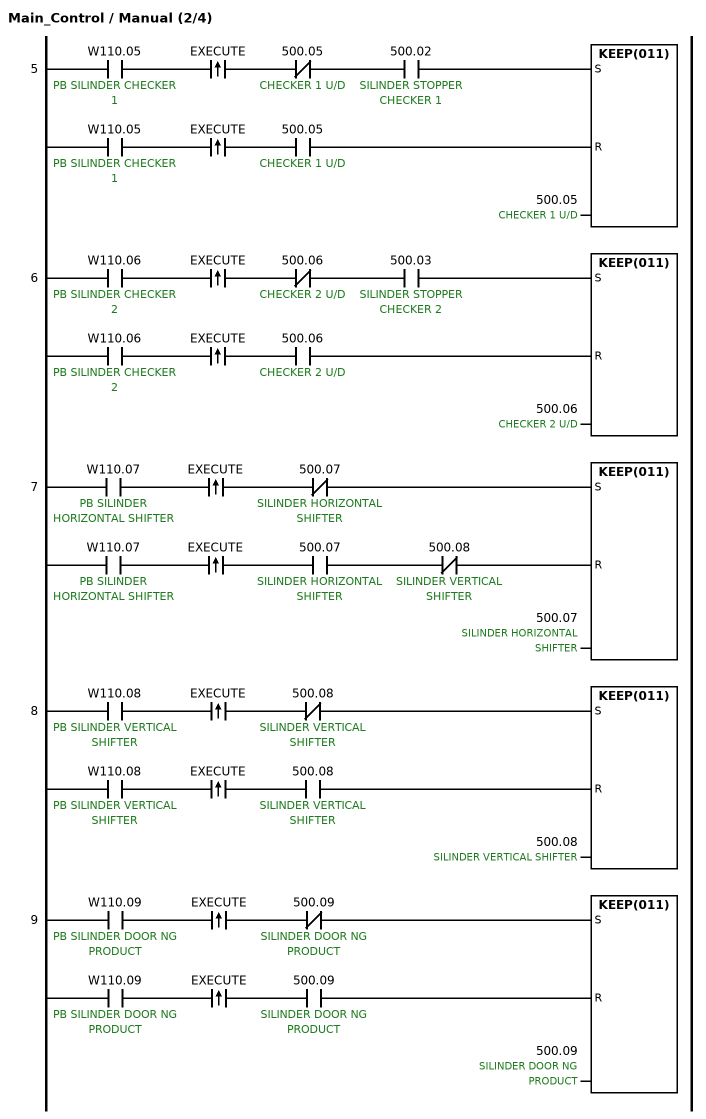
; rung 5
LD W110.05  ; PB SILINDER CHECKER 1
@AND EXECUTE
ANDNOT 500.05  ; CHECKER 1 U/D
AND 500.02  ; SILINDER STOPPER CHECKER 1
LD W110.05  ; PB SILINDER CHECKER 1
@AND EXECUTE
AND 500.05  ; CHECKER 1 U/D
KEEP(011) 500.05  ; CHECKER 1 U/D
; rung 6
LD W110.06  ; PB SILINDER CHECKER 2
@AND EXECUTE
ANDNOT 500.06  ; CHECKER 2 U/D
AND 500.03  ; SILINDER STOPPER CHECKER 2
LD W110.06  ; PB SILINDER CHECKER 2
@AND EXECUTE
AND 500.06  ; CHECKER 2 U/D
KEEP(011) 500.06  ; CHECKER 2 U/D
; rung 7
LD W110.07  ; PB SILINDER HORIZONTAL SHIFTER
@AND EXECUTE
ANDNOT 500.07  ; SILINDER HORIZONTAL SHIFTER
LD W110.07  ; PB SILINDER HORIZONTAL SHIFTER
@AND EXECUTE
AND 500.07  ; SILINDER HORIZONTAL SHIFTER
ANDNOT 500.08  ; SILINDER VERTICAL SHIFTER
KEEP(011) 500.07  ; SILINDER HORIZONTAL SHIFTER
; rung 8
LD W110.08  ; PB SILINDER VERTICAL SHIFTER
@AND EXECUTE
ANDNOT 500.08  ; SILINDER VERTICAL SHIFTER
LD W110.08  ; PB SILINDER VERTICAL SHIFTER
@AND EXECUTE
AND 500.08  ; SILINDER VERTICAL SHIFTER
KEEP(011) 500.08  ; SILINDER VERTICAL SHIFTER
; rung 9
LD W110.09  ; PB SILINDER DOOR NG PRODUCT
@AND EXECUTE
ANDNOT 500.09  ; SILINDER DOOR NG PRODUCT
LD W110.09  ; PB SILINDER DOOR NG PRODUCT
@AND EXECUTE
AND 500.09  ; SILINDER DOOR NG PRODUCT
KEEP(011) 500.09  ; SILINDER DOOR NG PRODUCT

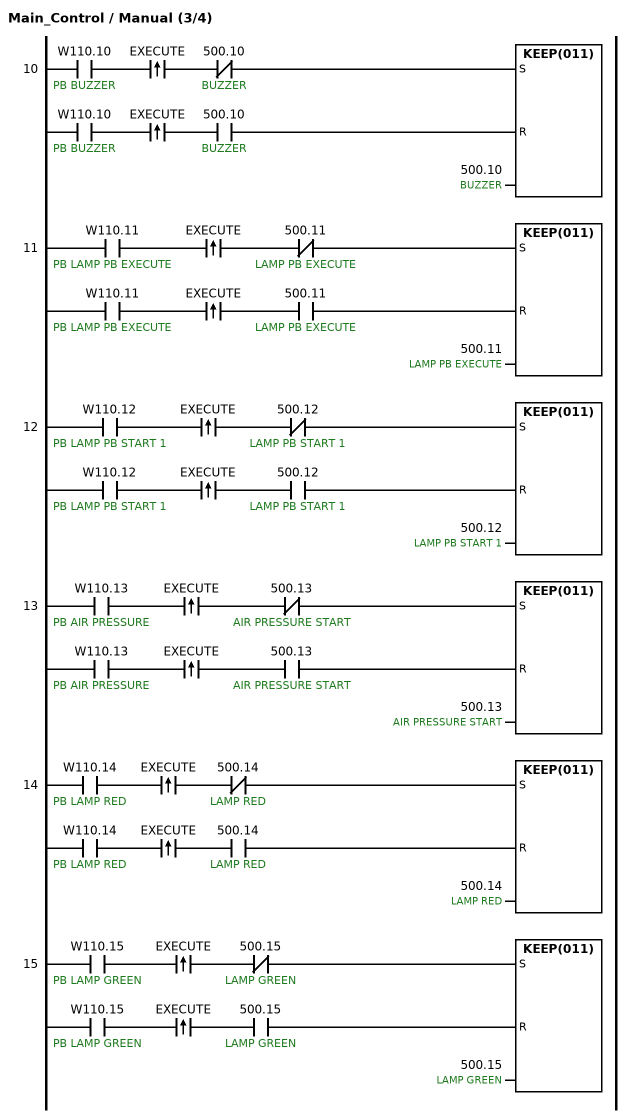
; rung 10
LD W110.10  ; PB BUZZER
@AND EXECUTE
ANDNOT 500.10  ; BUZZER
LD W110.10  ; PB BUZZER
@AND EXECUTE
AND 500.10  ; BUZZER
KEEP(011) 500.10  ; BUZZER
; rung 11
LD W110.11  ; PB LAMP PB EXECUTE
@AND EXECUTE
ANDNOT 500.11  ; LAMP PB EXECUTE
LD W110.11  ; PB LAMP PB EXECUTE
@AND EXECUTE
AND 500.11  ; LAMP PB EXECUTE
KEEP(011) 500.11  ; LAMP PB EXECUTE
; rung 12
LD W110.12  ; PB LAMP PB START 1
@AND EXECUTE
ANDNOT 500.12  ; LAMP PB START 1
LD W110.12  ; PB LAMP PB START 1
@AND EXECUTE
AND 500.12  ; LAMP PB START 1
KEEP(011) 500.12  ; LAMP PB START 1
; rung 13
LD W110.13  ; PB AIR PRESSURE
@AND EXECUTE
ANDNOT 500.13  ; AIR PRESSURE START
LD W110.13  ; PB AIR PRESSURE
@AND EXECUTE
AND 500.13  ; AIR PRESSURE START
KEEP(011) 500.13  ; AIR PRESSURE START
; rung 14
LD W110.14  ; PB LAMP RED
@AND EXECUTE
ANDNOT 500.14  ; LAMP RED
LD W110.14  ; PB LAMP RED
@AND EXECUTE
AND 500.14  ; LAMP RED
KEEP(011) 500.14  ; LAMP RED
; rung 15
LD W110.15  ; PB LAMP GREEN
@AND EXECUTE
ANDNOT 500.15  ; LAMP GREEN
LD W110.15  ; PB LAMP GREEN
@AND EXECUTE
AND 500.15  ; LAMP GREEN
KEEP(011) 500.15  ; LAMP GREEN

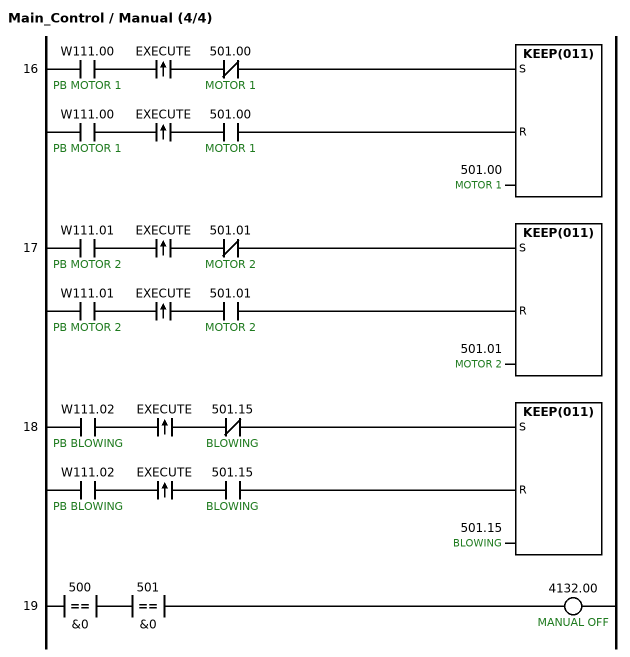
; rung 16
LD W111.00  ; PB MOTOR 1
@AND EXECUTE
ANDNOT 501.00  ; MOTOR 1
LD W111.00  ; PB MOTOR 1
@AND EXECUTE
AND 501.00  ; MOTOR 1
KEEP(011) 501.00  ; MOTOR 1
; rung 17
LD W111.01  ; PB MOTOR 2
@AND EXECUTE
ANDNOT 501.01  ; MOTOR 2
LD W111.01  ; PB MOTOR 2
@AND EXECUTE
AND 501.01  ; MOTOR 2
KEEP(011) 501.01  ; MOTOR 2
; rung 18
LD W111.02  ; PB BLOWING
@AND EXECUTE
ANDNOT 501.15  ; BLOWING
LD W111.02  ; PB BLOWING
@AND EXECUTE
AND 501.15  ; BLOWING
KEEP(011) 501.15  ; BLOWING
; rung 19
LD=(300) 500 &0
AND=(300) 501 &0
OUT 4132.00  ; MANUAL OFF

### Section Error

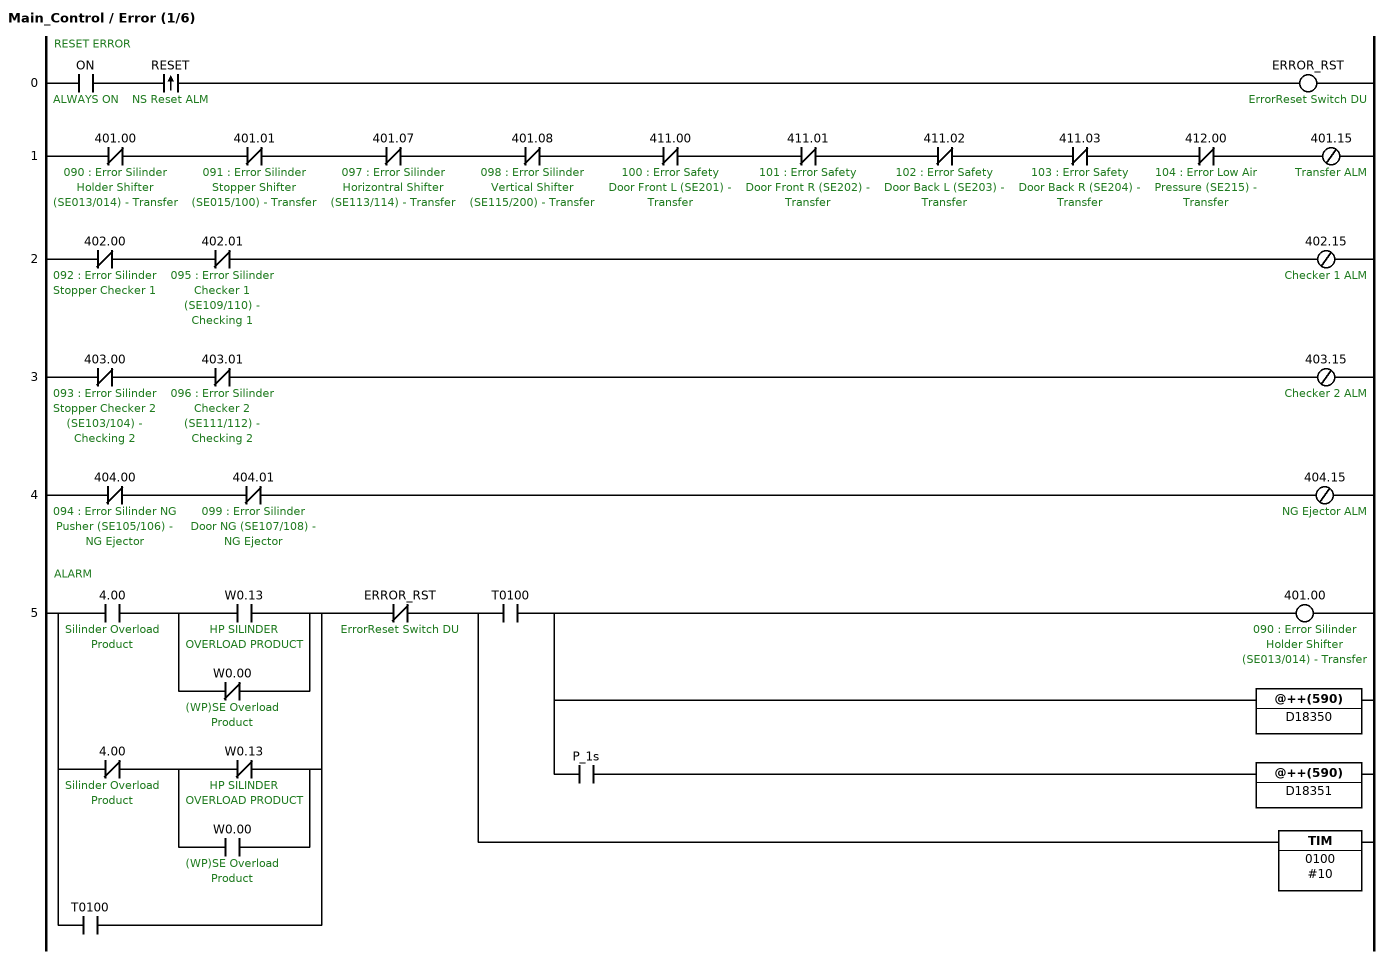
; rung 0: RESET ERROR
LD ON  ; ALWAYS ON
@AND RESET  ; NS Reset ALM
OUT ERROR_RST  ; ErrorReset Switch DU
; rung 1
LDNOT 401.00  ; 090 : Error Silinder Holder Shifter (SE013/014) - Transfer
ANDNOT 401.01  ; 091 : Error Silinder Stopper Shifter (SE015/100) - Transfer
ANDNOT 401.07  ; 097 : Error Silinder Horizontral Shifter (SE113/114) - Transfer
ANDNOT 401.08  ; 098 : Error Silinder Vertical Shifter (SE115/200) - Transfer
ANDNOT 411.00  ; 100 : Error Safety Door Front L (SE201) - Transfer
ANDNOT 411.01  ; 101 : Error Safety Door Front R (SE202) - Transfer
ANDNOT 411.02  ; 102 : Error Safety Door Back L (SE203) - Transfer
ANDNOT 411.03  ; 103 : Error Safety Door Back R (SE204) - Transfer
ANDNOT 412.00  ; 104 : Error Low Air Pressure (SE215) - Transfer
OUTNOT 401.15  ; Transfer ALM
; rung 2
LDNOT 402.00  ; 092 : Error Silinder Stopper Checker 1
ANDNOT 402.01  ; 095 : Error Silinder Checker 1 (SE109/110) - Checking 1
OUTNOT 402.15  ; Checker 1 ALM
; rung 3
LDNOT 403.00  ; 093 : Error Silinder Stopper Checker 2 (SE103/104) - Checking 2
ANDNOT 403.01  ; 096 : Error Silinder Checker 2 (SE111/112) - Checking 2
OUTNOT 403.15  ; Checker 2 ALM
; rung 4
LDNOT 404.00  ; 094 : Error Silinder NG Pusher (SE105/106) - NG Ejector
ANDNOT 404.01  ; 099 : Error Silinder Door NG (SE107/108) - NG Ejector
OUTNOT 404.15  ; NG Ejector ALM
; rung 5: ALARM
LD 4.00  ; Silinder Overload Product
LD W0.13  ; HP SILINDER OVERLOAD PRODUCT
ORNOT W0.00  ; (WP)SE Overload Product
ANDLD
LDNOT 4.00  ; Silinder Overload Product
LDNOT W0.13  ; HP SILINDER OVERLOAD PRODUCT
OR W0.00  ; (WP)SE Overload Product
ANDLD
ORLD
OR T0100
ANDNOT ERROR_RST  ; ErrorReset Switch DU
OUT TR0
AND T0100
OUT 401.00  ; 090 : Error Silinder Holder Shifter (SE013/014) - Transfer
@++(590) D18350
AND P_1s
@++(590) D18351
LD TR0
TIM 0100 #10

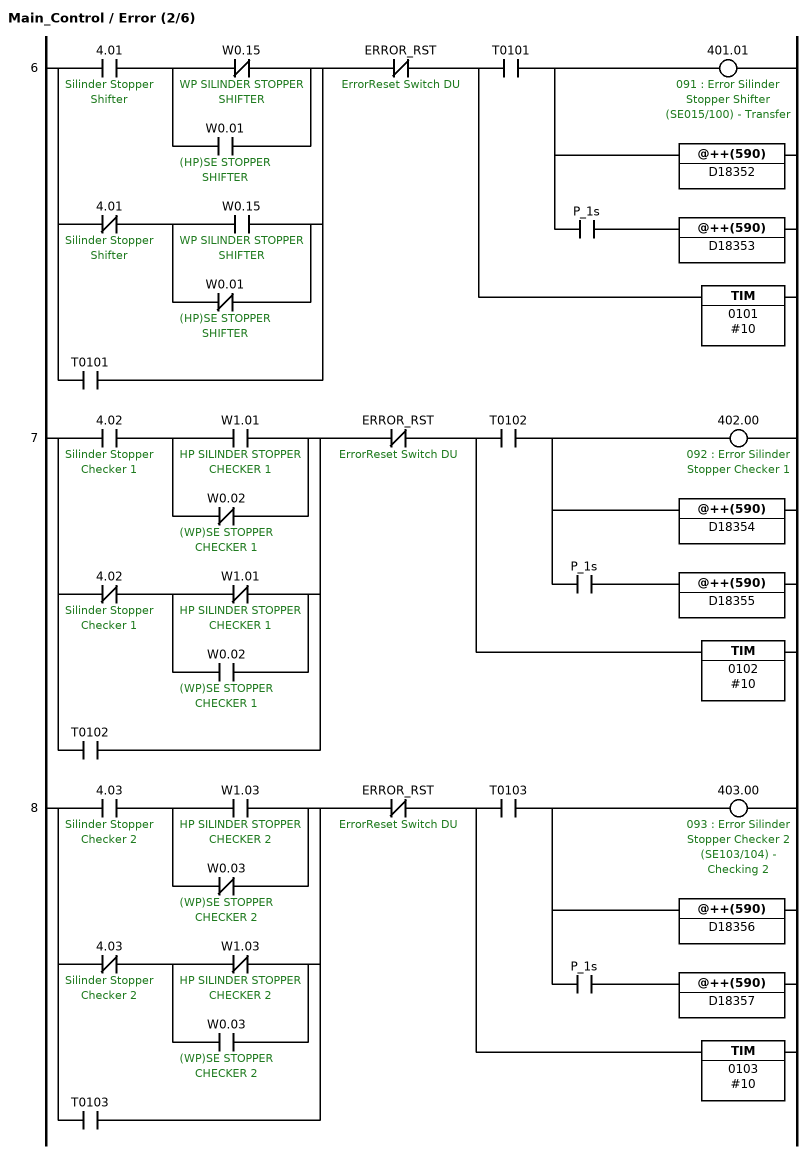
; rung 6
LD 4.01  ; Silinder Stopper Shifter
LDNOT W0.15  ; WP SILINDER STOPPER SHIFTER
OR W0.01  ; (HP)SE STOPPER SHIFTER
ANDLD
LDNOT 4.01  ; Silinder Stopper Shifter
LD W0.15  ; WP SILINDER STOPPER SHIFTER
ORNOT W0.01  ; (HP)SE STOPPER SHIFTER
ANDLD
ORLD
OR T0101
ANDNOT ERROR_RST  ; ErrorReset Switch DU
OUT TR0
AND T0101
OUT 401.01  ; 091 : Error Silinder Stopper Shifter (SE015/100) - Transfer
@++(590) D18352
AND P_1s
@++(590) D18353
LD TR0
TIM 0101 #10
; rung 7
LD 4.02  ; Silinder Stopper Checker 1
LD W1.01  ; HP SILINDER STOPPER CHECKER 1
ORNOT W0.02  ; (WP)SE STOPPER CHECKER 1
ANDLD
LDNOT 4.02  ; Silinder Stopper Checker 1
LDNOT W1.01  ; HP SILINDER STOPPER CHECKER 1
OR W0.02  ; (WP)SE STOPPER CHECKER 1
ANDLD
ORLD
OR T0102
ANDNOT ERROR_RST  ; ErrorReset Switch DU
OUT TR0
AND T0102
OUT 402.00  ; 092 : Error Silinder Stopper Checker 1
@++(590) D18354
AND P_1s
@++(590) D18355
LD TR0
TIM 0102 #10
; rung 8
LD 4.03  ; Silinder Stopper Checker 2
LD W1.03  ; HP SILINDER STOPPER CHECKER 2
ORNOT W0.03  ; (WP)SE STOPPER CHECKER 2
ANDLD
LDNOT 4.03  ; Silinder Stopper Checker 2
LDNOT W1.03  ; HP SILINDER STOPPER CHECKER 2
OR W0.03  ; (WP)SE STOPPER CHECKER 2
ANDLD
ORLD
OR T0103
ANDNOT ERROR_RST  ; ErrorReset Switch DU
OUT TR0
AND T0103
OUT 403.00  ; 093 : Error Silinder Stopper Checker 2 (SE103/104) - Checking 2
@++(590) D18356
AND P_1s
@++(590) D18357
LD TR0
TIM 0103 #10

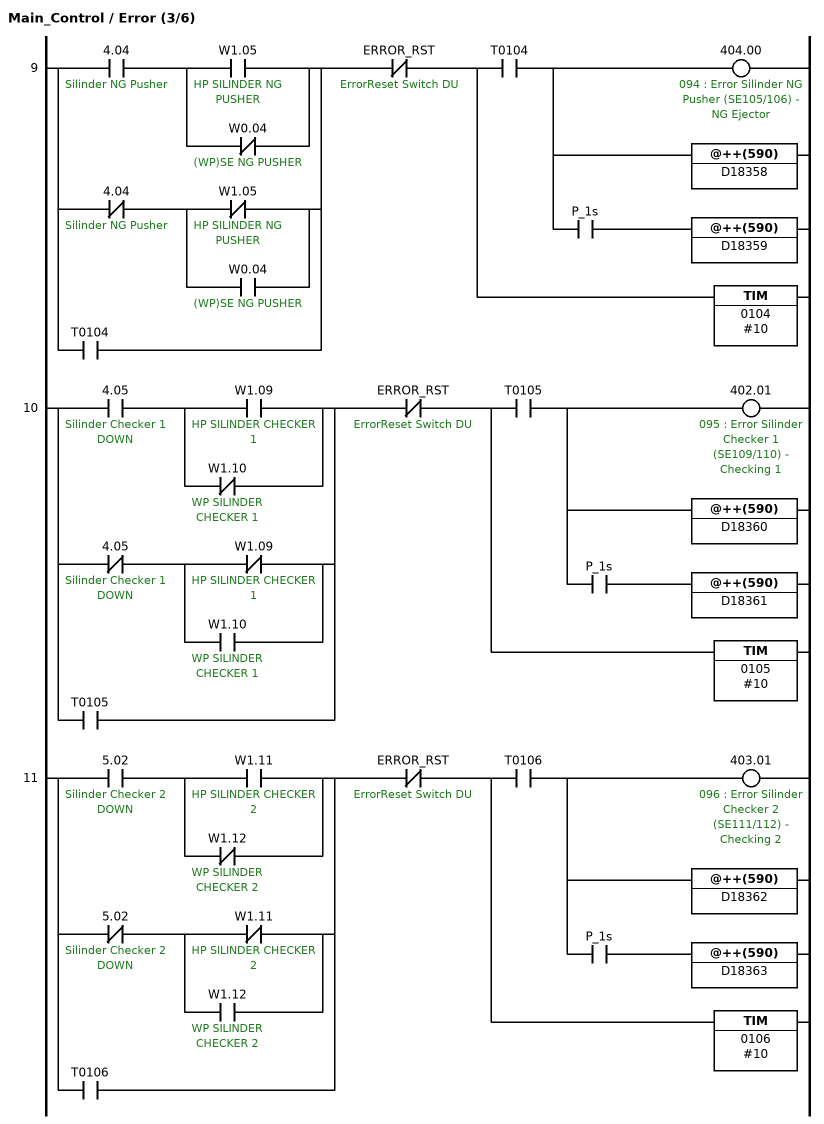
; rung 9
LD 4.04  ; Silinder NG Pusher
LD W1.05  ; HP SILINDER NG PUSHER
ORNOT W0.04  ; (WP)SE NG PUSHER
ANDLD
LDNOT 4.04  ; Silinder NG Pusher
LDNOT W1.05  ; HP SILINDER NG PUSHER
OR W0.04  ; (WP)SE NG PUSHER
ANDLD
ORLD
OR T0104
ANDNOT ERROR_RST  ; ErrorReset Switch DU
OUT TR0
AND T0104
OUT 404.00  ; 094 : Error Silinder NG Pusher (SE105/106) - NG Ejector
@++(590) D18358
AND P_1s
@++(590) D18359
LD TR0
TIM 0104 #10
; rung 10
LD 4.05  ; Silinder Checker 1 DOWN
LD W1.09  ; HP SILINDER CHECKER 1
ORNOT W1.10  ; WP SILINDER CHECKER 1
ANDLD
LDNOT 4.05  ; Silinder Checker 1 DOWN
LDNOT W1.09  ; HP SILINDER CHECKER 1
OR W1.10  ; WP SILINDER CHECKER 1
ANDLD
ORLD
OR T0105
ANDNOT ERROR_RST  ; ErrorReset Switch DU
OUT TR0
AND T0105
OUT 402.01  ; 095 : Error Silinder Checker 1 (SE109/110) - Checking 1
@++(590) D18360
AND P_1s
@++(590) D18361
LD TR0
TIM 0105 #10
; rung 11
LD 5.02  ; Silinder Checker 2 DOWN
LD W1.11  ; HP SILINDER CHECKER 2
ORNOT W1.12  ; WP SILINDER CHECKER 2
ANDLD
LDNOT 5.02  ; Silinder Checker 2 DOWN
LDNOT W1.11  ; HP SILINDER CHECKER 2
OR W1.12  ; WP SILINDER CHECKER 2
ANDLD
ORLD
OR T0106
ANDNOT ERROR_RST  ; ErrorReset Switch DU
OUT TR0
AND T0106
OUT 403.01  ; 096 : Error Silinder Checker 2 (SE111/112) - Checking 2
@++(590) D18362
AND P_1s
@++(590) D18363
LD TR0
TIM 0106 #10

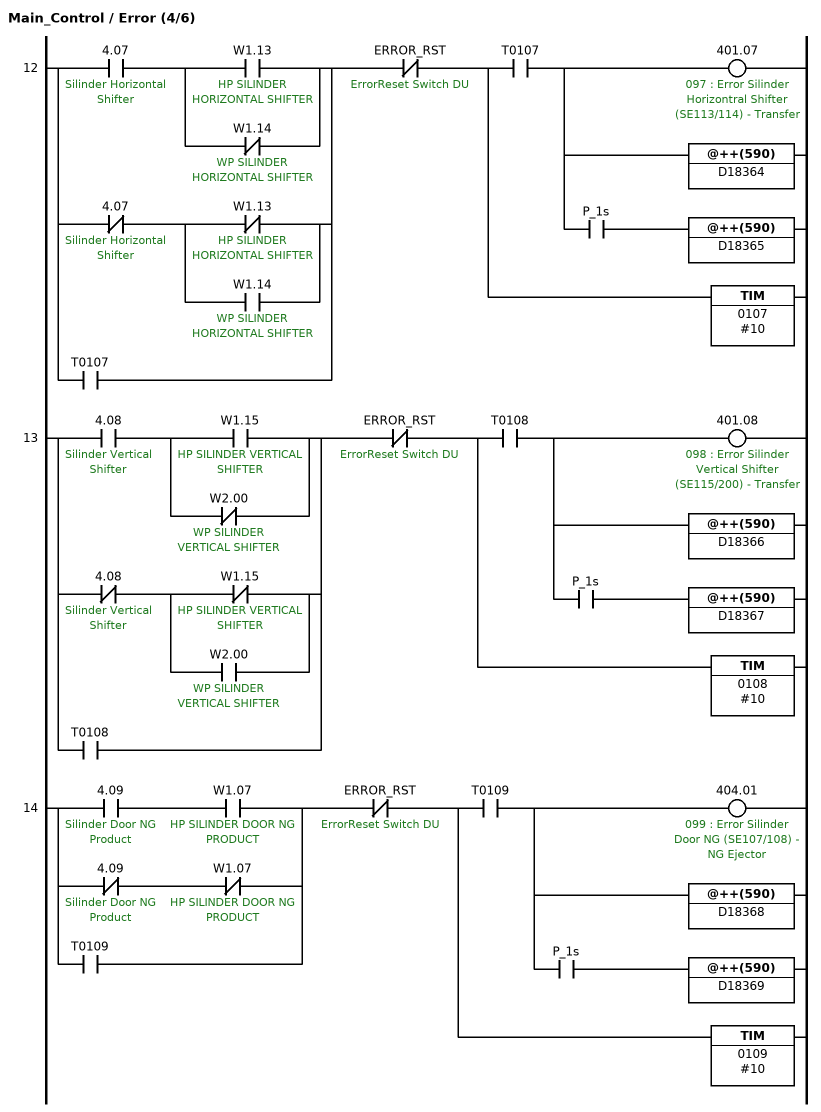
; rung 12
LD 4.07  ; Silinder Horizontal Shifter
LD W1.13  ; HP SILINDER HORIZONTAL SHIFTER
ORNOT W1.14  ; WP SILINDER HORIZONTAL SHIFTER
ANDLD
LDNOT 4.07  ; Silinder Horizontal Shifter
LDNOT W1.13  ; HP SILINDER HORIZONTAL SHIFTER
OR W1.14  ; WP SILINDER HORIZONTAL SHIFTER
ANDLD
ORLD
OR T0107
ANDNOT ERROR_RST  ; ErrorReset Switch DU
OUT TR0
AND T0107
OUT 401.07  ; 097 : Error Silinder Horizontral Shifter (SE113/114) - Transfer
@++(590) D18364
AND P_1s
@++(590) D18365
LD TR0
TIM 0107 #10
; rung 13
LD 4.08  ; Silinder Vertical Shifter
LD W1.15  ; HP SILINDER VERTICAL SHIFTER
ORNOT W2.00  ; WP SILINDER VERTICAL SHIFTER
ANDLD
LDNOT 4.08  ; Silinder Vertical Shifter
LDNOT W1.15  ; HP SILINDER VERTICAL SHIFTER
OR W2.00  ; WP SILINDER VERTICAL SHIFTER
ANDLD
ORLD
OR T0108
ANDNOT ERROR_RST  ; ErrorReset Switch DU
OUT TR0
AND T0108
OUT 401.08  ; 098 : Error Silinder Vertical Shifter (SE115/200) - Transfer
@++(590) D18366
AND P_1s
@++(590) D18367
LD TR0
TIM 0108 #10
; rung 14
LD 4.09  ; Silinder Door NG Product
AND W1.07  ; HP SILINDER DOOR NG PRODUCT
LDNOT 4.09  ; Silinder Door NG Product
ANDNOT W1.07  ; HP SILINDER DOOR NG PRODUCT
ORLD
OR T0109
ANDNOT ERROR_RST  ; ErrorReset Switch DU
OUT TR0
AND T0109
OUT 404.01  ; 099 : Error Silinder Door NG (SE107/108) - NG Ejector
@++(590) D18368
AND P_1s
@++(590) D18369
LD TR0
TIM 0109 #10

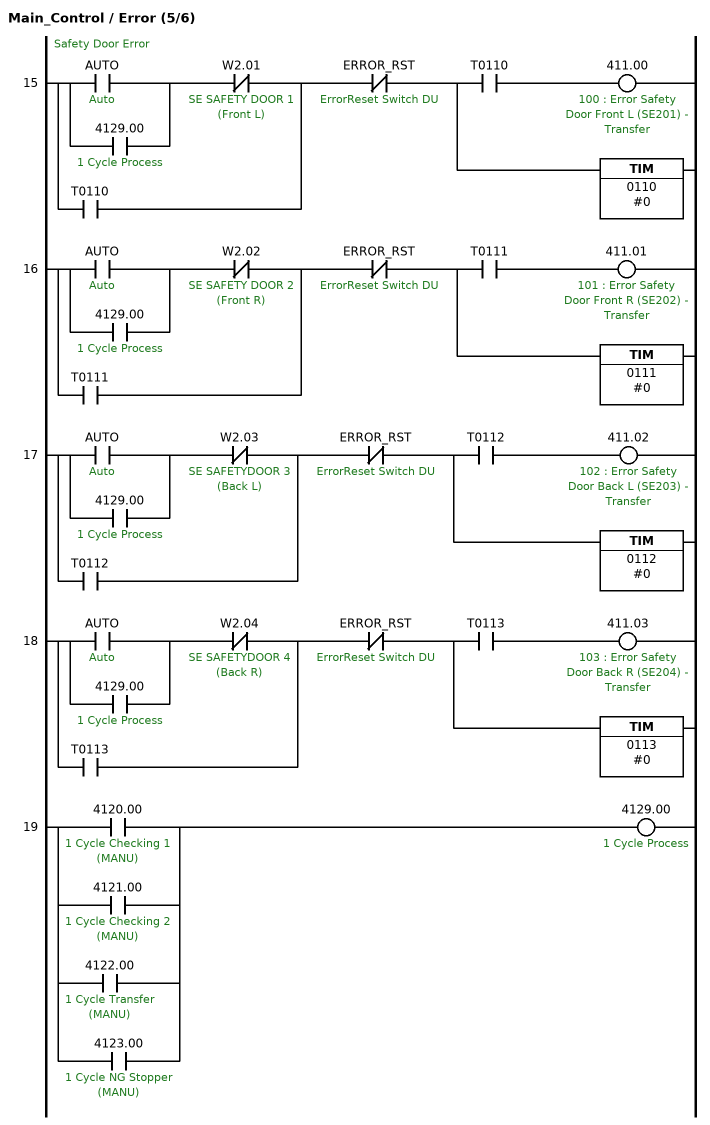
; rung 15: Safety Door Error
LD AUTO  ; Auto
OR 4129.00  ; 1 Cycle Process
ANDNOT W2.01  ; SE SAFETY DOOR 1 (Front L)
OR T0110
ANDNOT ERROR_RST  ; ErrorReset Switch DU
OUT TR0
AND T0110
OUT 411.00  ; 100 : Error Safety Door Front L (SE201) - Transfer
LD TR0
TIM 0110 #0
; rung 16
LD AUTO  ; Auto
OR 4129.00  ; 1 Cycle Process
ANDNOT W2.02  ; SE SAFETY DOOR 2 (Front R)
OR T0111
ANDNOT ERROR_RST  ; ErrorReset Switch DU
OUT TR0
AND T0111
OUT 411.01  ; 101 : Error Safety Door Front R (SE202) - Transfer
LD TR0
TIM 0111 #0
; rung 17
LD AUTO  ; Auto
OR 4129.00  ; 1 Cycle Process
ANDNOT W2.03  ; SE SAFETYDOOR 3 (Back L)
OR T0112
ANDNOT ERROR_RST  ; ErrorReset Switch DU
OUT TR0
AND T0112
OUT 411.02  ; 102 : Error Safety Door Back L (SE203) - Transfer
LD TR0
TIM 0112 #0
; rung 18
LD AUTO  ; Auto
OR 4129.00  ; 1 Cycle Process
ANDNOT W2.04  ; SE SAFETYDOOR 4 (Back R)
OR T0113
ANDNOT ERROR_RST  ; ErrorReset Switch DU
OUT TR0
AND T0113
OUT 411.03  ; 103 : Error Safety Door Back R (SE204) - Transfer
LD TR0
TIM 0113 #0
; rung 19
LD 4120.00  ; 1 Cycle Checking 1 (MANU)
OR 4121.00  ; 1 Cycle Checking 2 (MANU)
OR 4122.00  ; 1 Cycle Transfer (MANU)
OR 4123.00  ; 1 Cycle NG Stopper (MANU)
OUT 4129.00  ; 1 Cycle Process

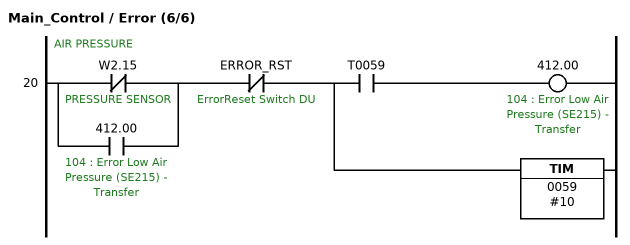
; rung 20: AIR PRESSURE
LDNOT W2.15  ; PRESSURE SENSOR
OR 412.00  ; 104 : Error Low Air Pressure (SE215) - Transfer
ANDNOT ERROR_RST  ; ErrorReset Switch DU
OUT TR0
AND T0059
OUT 412.00  ; 104 : Error Low Air Pressure (SE215) - Transfer
LD TR0
TIM 0059 #10

### Section Auto_Run

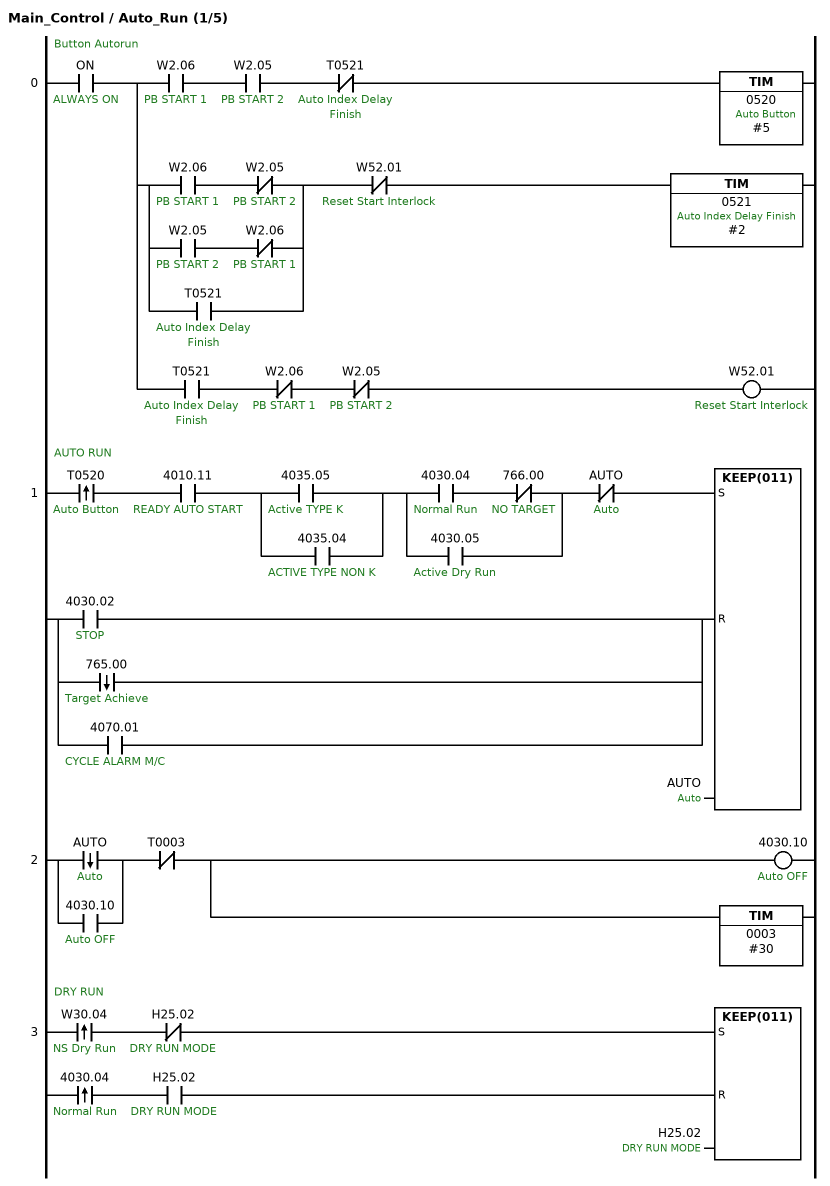
; rung 0: Button Autorun
LD ON  ; ALWAYS ON
OUT TR0
AND W2.06  ; PB START 1
AND W2.05  ; PB START 2
ANDNOT T0521  ; Auto Index Delay Finish
TIM 0520 #5  ; Auto Button
LD TR0
LD W2.06  ; PB START 1
ANDNOT W2.05  ; PB START 2
LD W2.05  ; PB START 2
ANDNOT W2.06  ; PB START 1
ORLD
OR T0521  ; Auto Index Delay Finish
ANDLD
ANDNOT W52.01  ; Reset Start Interlock
TIM 0521 #2  ; Auto Index Delay Finish
LD TR0
AND T0521  ; Auto Index Delay Finish
ANDNOT W2.06  ; PB START 1
ANDNOT W2.05  ; PB START 2
OUT W52.01  ; Reset Start Interlock
; rung 1: AUTO RUN
@LD T0520  ; Auto Button
AND 4010.11  ; READY AUTO START
LD 4035.05  ; Active TYPE K
OR 4035.04  ; ACTIVE TYPE NON K
ANDLD
LD 4030.04  ; Normal Run
ANDNOT 766.00  ; NO TARGET
OR 4030.05  ; Active Dry Run
ANDLD
ANDNOT AUTO  ; Auto
LD 4030.02  ; STOP
%OR 765.00  ; Target Achieve
OR 4070.01  ; CYCLE ALARM M/C
KEEP(011) AUTO  ; Auto
; rung 2
%LD AUTO  ; Auto
OR 4030.10  ; Auto OFF
ANDNOT T0003
OUT 4030.10  ; Auto OFF
TIM 0003 #30
; rung 3: DRY RUN
@LD W30.04  ; NS Dry Run
ANDNOT H25.02  ; DRY RUN MODE
@LD 4030.04  ; Normal Run
AND H25.02  ; DRY RUN MODE
KEEP(011) H25.02  ; DRY RUN MODE

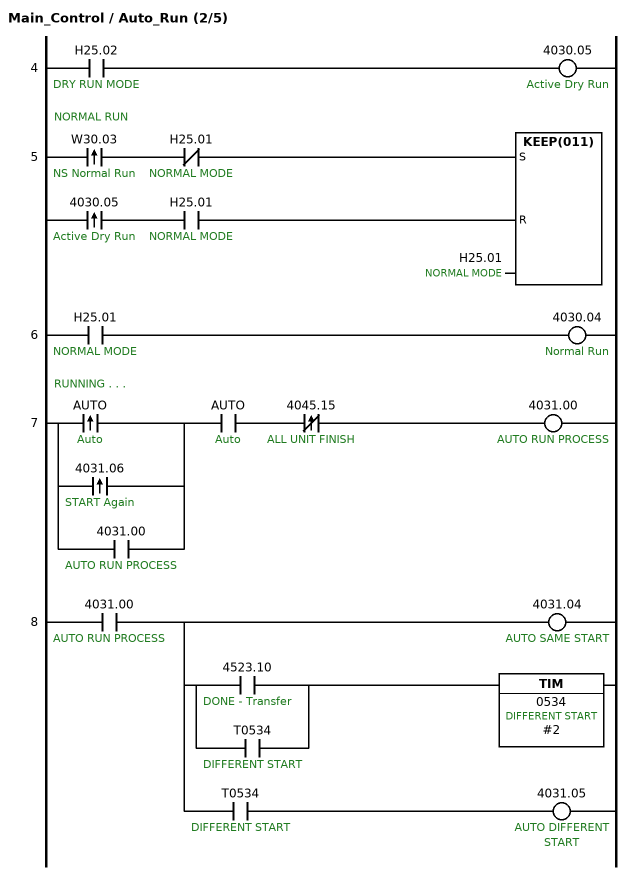
; rung 4
LD H25.02  ; DRY RUN MODE
OUT 4030.05  ; Active Dry Run
; rung 5: NORMAL RUN
@LD W30.03  ; NS Normal Run
ANDNOT H25.01  ; NORMAL MODE
@LD 4030.05  ; Active Dry Run
AND H25.01  ; NORMAL MODE
KEEP(011) H25.01  ; NORMAL MODE
; rung 6
LD H25.01  ; NORMAL MODE
OUT 4030.04  ; Normal Run
; rung 7: RUNNING . . .
@LD AUTO  ; Auto
@OR 4031.06  ; START Again
OR 4031.00  ; AUTO RUN PROCESS
AND AUTO  ; Auto
@ANDNOT 4045.15  ; ALL UNIT FINISH
OUT 4031.00  ; AUTO RUN PROCESS
; rung 8
LD 4031.00  ; AUTO RUN PROCESS
OUT TR0
OUT 4031.04  ; AUTO SAME START
LD 4523.10  ; DONE - Transfer
OR T0534  ; DIFFERENT START
ANDLD
TIM 0534 #2  ; DIFFERENT START
LD TR0
AND T0534  ; DIFFERENT START
OUT 4031.05  ; AUTO DIFFERENT START

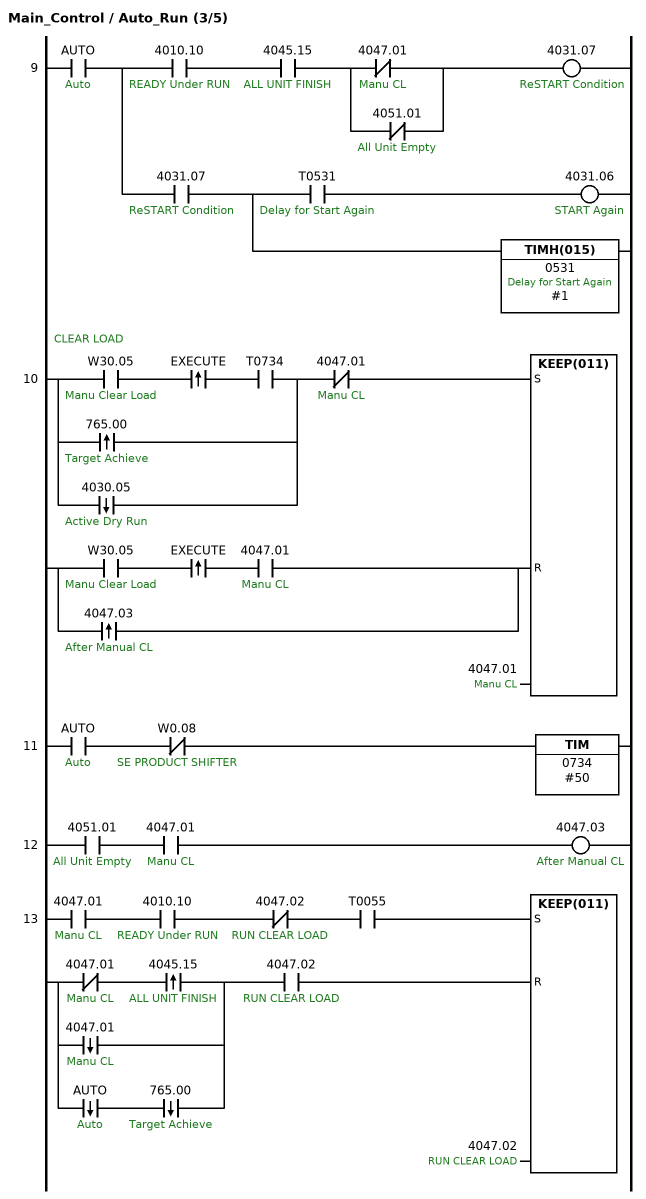
; rung 9
LD AUTO  ; Auto
OUT TR0
AND 4010.10  ; READY Under RUN
AND 4045.15  ; ALL UNIT FINISH
LDNOT 4047.01  ; Manu CL
ORNOT 4051.01  ; All Unit Empty
ANDLD
OUT 4031.07  ; ReSTART Condition
LD TR0
AND 4031.07  ; ReSTART Condition
OUT TR0
AND T0531  ; Delay for Start Again
OUT 4031.06  ; START Again
LD TR0
TIMH(015) 0531 #1  ; Delay for Start Again
; rung 10: CLEAR LOAD
LD W30.05  ; Manu Clear Load
@AND EXECUTE
AND T0734
@OR 765.00  ; Target Achieve
%OR 4030.05  ; Active Dry Run
ANDNOT 4047.01  ; Manu CL
LD W30.05  ; Manu Clear Load
@AND EXECUTE
AND 4047.01  ; Manu CL
@OR 4047.03  ; After Manual CL
KEEP(011) 4047.01  ; Manu CL
; rung 11
LD AUTO  ; Auto
ANDNOT W0.08  ; SE PRODUCT SHIFTER
TIM 0734 #50
; rung 12
LD 4051.01  ; All Unit Empty
AND 4047.01  ; Manu CL
OUT 4047.03  ; After Manual CL
; rung 13
LD 4047.01  ; Manu CL
AND 4010.10  ; READY Under RUN
ANDNOT 4047.02  ; RUN CLEAR LOAD
AND T0055
LDNOT 4047.01  ; Manu CL
@AND 4045.15  ; ALL UNIT FINISH
%OR 4047.01  ; Manu CL
%LD AUTO  ; Auto
%AND 765.00  ; Target Achieve
ORLD
AND 4047.02  ; RUN CLEAR LOAD
KEEP(011) 4047.02  ; RUN CLEAR LOAD

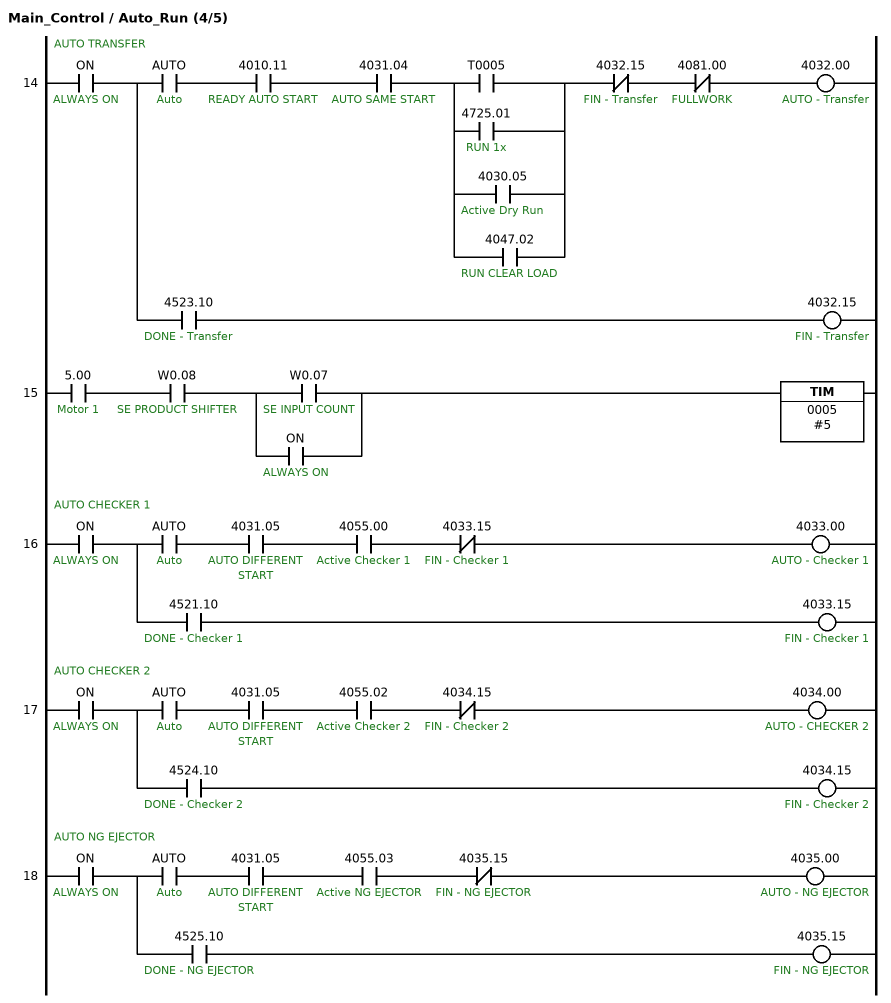
; rung 14: AUTO TRANSFER
LD ON  ; ALWAYS ON
OUT TR0
AND AUTO  ; Auto
AND 4010.11  ; READY AUTO START
AND 4031.04  ; AUTO SAME START
LD T0005
OR 4725.01  ; RUN 1x
OR 4030.05  ; Active Dry Run
OR 4047.02  ; RUN CLEAR LOAD
ANDLD
ANDNOT 4032.15  ; FIN - Transfer
ANDNOT 4081.00  ; FULLWORK
OUT 4032.00  ; AUTO - Transfer
LD TR0
AND 4523.10  ; DONE - Transfer
OUT 4032.15  ; FIN - Transfer
; rung 15
LD 5.00  ; Motor 1
AND W0.08  ; SE PRODUCT SHIFTER
LD W0.07  ; SE INPUT COUNT
OR ON  ; ALWAYS ON
ANDLD
TIM 0005 #5
; rung 16: AUTO CHECKER 1
LD ON  ; ALWAYS ON
OUT TR0
AND AUTO  ; Auto
AND 4031.05  ; AUTO DIFFERENT START
AND 4055.00  ; Active Checker 1
ANDNOT 4033.15  ; FIN - Checker 1
OUT 4033.00  ; AUTO - Checker 1
LD TR0
AND 4521.10  ; DONE - Checker 1
OUT 4033.15  ; FIN - Checker 1
; rung 17: AUTO CHECKER 2
LD ON  ; ALWAYS ON
OUT TR0
AND AUTO  ; Auto
AND 4031.05  ; AUTO DIFFERENT START
AND 4055.02  ; Active Checker 2
ANDNOT 4034.15  ; FIN - Checker 2
OUT 4034.00  ; AUTO - CHECKER 2
LD TR0
AND 4524.10  ; DONE - Checker 2
OUT 4034.15  ; FIN - Checker 2
; rung 18: AUTO NG EJECTOR
LD ON  ; ALWAYS ON
OUT TR0
AND AUTO  ; Auto
AND 4031.05  ; AUTO DIFFERENT START
AND 4055.03  ; Active NG EJECTOR
ANDNOT 4035.15  ; FIN - NG EJECTOR
OUT 4035.00  ; AUTO - NG EJECTOR
LD TR0
AND 4525.10  ; DONE - NG EJECTOR
OUT 4035.15  ; FIN - NG EJECTOR

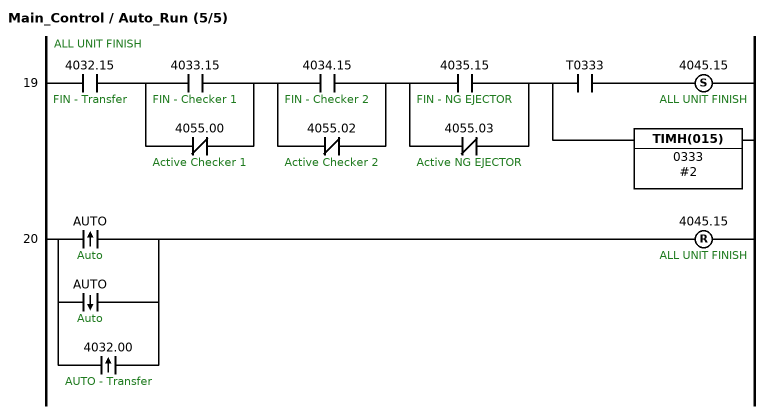
; rung 19: ALL UNIT FINISH
LD 4032.15  ; FIN - Transfer
LD 4033.15  ; FIN - Checker 1
ORNOT 4055.00  ; Active Checker 1
ANDLD
LD 4034.15  ; FIN - Checker 2
ORNOT 4055.02  ; Active Checker 2
ANDLD
LD 4035.15  ; FIN - NG EJECTOR
ORNOT 4055.03  ; Active NG EJECTOR
ANDLD
OUT TR0
AND T0333
SET 4045.15  ; ALL UNIT FINISH
LD TR0
TIMH(015) 0333 #2
; rung 20
@LD AUTO  ; Auto
%OR AUTO  ; Auto
@OR 4032.00  ; AUTO - Transfer
RSET 4045.15  ; ALL UNIT FINISH

### Section Process

